LIN {X 50.548,Y -47.576,Z -199.936,A -90.000,B 90.000,C 0.000} C_DIS
LIN {X 49.783,Y -47.603,Z -202.584,A -90.000,B 90.000,C 0.000} C_DIS
LIN {X 49.593,Y -47.607,Z -203.194,A -90.000,B 90.000,C 0.000} C_DIS
LIN {X 48.332,Y -47.644,Z -207.156,A -90.000,B 90.000,C 0.000} C_DIS
LIN {X 47.582,Y -47.662,Z -209.460,A -90.000,B 90.000,C 0.000} C_DIS
LIN {X 47.233,Y -47.673,Z -210.498,A -90.000,B 90.000,C 0.000} C_DIS
LIN {X 46.703,Y -47.673,Z -212.067,A -90.000,B 90.000,C 0.000} C_DIS
LIN {X 46.008,Y -47.674,Z -214.062,A -90.000,B 90.000,C 0.000} C_DIS
LIN {X 45.274,Y -47.666,Z -216.296,A -90.000,B 90.000,C 0.000} C_DIS
LIN {X 44.970,Y -47.666,Z -217.223,A -90.000,B 90.000,C 0.000} C_DIS
LIN {X 44.923,Y -47.667,Z -217.335,A -90.000,B 90.000,C 0.000} C_DIS
LIN {X 44.486,Y -47.667,Z -218.383,A -90.000,B 90.000,C 0.000} C_DIS
LIN {X 43.526,Y -47.657,Z -220.833,A -90.000,B 90.000,C 0.000} C_DIS
LIN {X 42.934,Y -47.657,Z -222.345,A -90.000,B 90.000,C 0.000} C_DIS
LIN {X 42.807,Y -47.663,Z -222.577,A -90.000,B 90.000,C 0.000} C_DIS
LIN {X 42.638,Y -47.663,Z -222.882,A -90.000,B 90.000,C 0.000} C_DIS
LIN {X 41.300,Y -47.652,Z -225.431,A -90.000,B 90.000,C 0.000} C_DIS
LIN {X 40.291,Y -47.650,Z -227.357,A -90.000,B 90.000,C 0.000} C_DIS
LIN {X 40.021,Y -47.664,Z -227.703,A -90.000,B 90.000,C 0.000} C_DIS
LIN {X 39.850,Y -47.667,Z -227.921,A -90.000,B 90.000,C 0.000} C_DIS
LIN {X 37.302,Y -47.652,Z -231.289,A -90.000,B 90.000,C 0.000} C_DIS
LIN {X 36.746,Y -47.651,Z -232.025,A -90.000,B 90.000,C 0.000} C_DIS
LIN {X 36.686,Y -47.653,Z -232.080,A -90.000,B 90.000,C 0.000} C_DIS
LIN {X 36.061,Y -47.684,Z -232.614,A -90.000,B 90.000,C 0.000} C_DIS
LIN {X 35.829,Y -47.686,Z -232.809,A -90.000,B 90.000,C 0.000} C_DIS
LIN {X 35.506,Y -47.686,Z -233.081,A -90.000,B 90.000,C 0.000} C_DIS
LIN {X 34.289,Y -47.685,Z -234.104,A -90.000,B 90.000,C 0.000} C_DIS
LIN {X 33.544,Y -47.662,Z -234.725,A -90.000,B 90.000,C 0.000} C_DIS
LIN {X 31.821,Y -47.603,Z -236.201,A -90.000,B 90.000,C 0.000} C_DIS
LIN {X 31.643,Y -47.599,Z -236.332,A -90.000,B 90.000,C 0.000} C_DIS
LIN {X 30.851,Y -47.588,Z -236.838,A -90.000,B 90.000,C 0.000} C_DIS
LIN {X 30.642,Y -47.585,Z -236.965,A -90.000,B 90.000,C 0.000} C_DIS
LIN {X 29.999,Y -47.565,Z -237.355,A -90.000,B 90.000,C 0.000} C_DIS
LIN {X 26.309,Y -47.565,Z -238.632,A -90.000,B 90.000,C 0.000} C_DIS
LIN {X 26.101,Y -47.561,Z -238.703,A -90.000,B 90.000,C 0.000} C_DIS
LIN {X 25.572,Y -47.541,Z -238.883,A -90.000,B 90.000,C 0.000} C_DIS
LIN {X 24.943,Y -47.512,Z -239.098,A -90.000,B 90.000,C 0.000} C_DIS
LIN {X 24.543,Y -47.495,Z -239.210,A -90.000,B 90.000,C 0.000} C_DIS
LIN {X 24.462,Y -47.492,Z -239.233,A -90.000,B 90.000,C 0.000} C_DIS
LIN {X 24.387,Y -47.494,Z -239.257,A -90.000,B 90.000,C 0.000} C_DIS
LIN {X 24.313,Y -47.492,Z -239.283,A -90.000,B 90.000,C 0.000} C_DIS
LIN {X 24.239,Y -47.490,Z -239.311,A -90.000,B 90.000,C 0.000} C_DIS
LIN {X 24.093,Y -47.485,Z -239.376,A -90.000,B 90.000,C 0.000} C_DIS
LIN {X 23.947,Y -47.481,Z -239.382,A -90.000,B 90.000,C 0.000} C_DIS
LIN {X 23.875,Y -47.479,Z -239.388,A -90.000,B 90.000,C 0.000} C_DIS
LIN {X 23.732,Y -47.475,Z -239.409,A -90.000,B 90.000,C 0.000} C_DIS
LIN {X 23.592,Y -47.471,Z -239.439,A -90.000,B 90.000,C 0.000} C_DIS
LIN {X 23.385,Y -47.464,Z -239.496,A -90.000,B 90.000,C 0.000} C_DIS
LIN {X 23.249,Y -47.459,Z -239.542,A -90.000,B 90.000,C 0.000} C_DIS
LIN {X 23.115,Y -47.453,Z -239.594,A -90.000,B 90.000,C 0.000} C_DIS
LIN {X 22.916,Y -47.444,Z -239.681,A -90.000,B 90.000,C 0.000} C_DIS
LIN {X 22.655,Y -47.432,Z -239.810,A -90.000,B 90.000,C 0.000} C_DIS
LIN {X 22.008,Y -47.400,Z -240.160,A -90.000,B 90.000,C 0.000} C_DIS
LIN {X 21.748,Y -47.387,Z -240.295,A -90.000,B 90.000,C 0.000} C_DIS
LIN {X 21.484,Y -47.375,Z -240.419,A -90.000,B 90.000,C 0.000} C_DIS
LIN {X 21.350,Y -47.368,Z -240.477,A -90.000,B 90.000,C 0.000} C_DIS
LIN {X 21.215,Y -47.362,Z -240.528,A -90.000,B 90.000,C 0.000} C_DIS
LIN {X 21.078,Y -47.356,Z -240.571,A -90.000,B 90.000,C 0.000} C_DIS
LIN {X 21.009,Y -47.353,Z -240.590,A -90.000,B 90.000,C 0.000} C_DIS
LIN {X 20.940,Y -47.350,Z -240.606,A -90.000,B 90.000,C 0.000} C_DIS
LIN {X 20.839,Y -47.345,Z -240.621,A -90.000,B 90.000,C 0.000} C_DIS
LIN {X 20.661,Y -47.337,Z -240.664,A -90.000,B 90.000,C 0.000} C_DIS
LIN {X 20.513,Y -47.331,Z -240.694,A -90.000,B 90.000,C 0.000} C_DIS
LIN {X 20.361,Y -47.324,Z -240.716,A -90.000,B 90.000,C 0.000} C_DIS
LIN {X 20.284,Y -47.321,Z -240.723,A -90.000,B 90.000,C 0.000} C_DIS
LIN {X 20.127,Y -47.314,Z -240.729,A -90.000,B 90.000,C 0.000} C_DIS
LIN {X 20.049,Y -47.308,Z -240.727,A -90.000,B 90.000,C 0.000} C_DIS
LIN {X 19.691,Y -47.308,Z -240.706,A -90.000,B 90.000,C 0.000} C_DIS
LIN {X 19.298,Y -47.308,Z -240.660,A -90.000,B 90.000,C 0.000} C_DIS
LIN {X 19.221,Y -47.308,Z -240.617,A -90.000,B 90.000,C 0.000} C_DIS
LIN {X 17.099,Y -47.308,Z -237.044,A -90.000,B 90.000,C 0.000} C_DIS
LIN {X 17.057,Y -47.308,Z -236.966,A -90.000,B 90.000,C 0.000} C_DIS
LIN {X 17.047,Y -47.308,Z -236.943,A -90.000,B 90.000,C 0.000} C_DIS
LIN {X 16.984,Y -47.308,Z -236.487,A -90.000,B 90.000,C 0.000} C_DIS
LIN {X 16.973,Y -47.308,Z -236.308,A -90.000,B 90.000,C 0.000} C_DIS
LIN {X 17.928,Y -47.308,Z -231.443,A -90.000,B 90.000,C 0.000} C_DIS
LIN {X 17.967,Y -47.308,Z -231.268,A -90.000,B 90.000,C 0.000} C_DIS
LIN {X 19.365,Y -47.308,Z -226.787,A -90.000,B 90.000,C 0.000} C_DIS
LIN {X 19.696,Y -47.308,Z -226.007,A -90.000,B 90.000,C 0.000} C_DIS
LIN {X 20.442,Y -47.308,Z -224.463,A -90.000,B 90.000,C 0.000} C_DIS
LIN {X 22.215,Y -47.308,Z -221.029,A -90.000,B 90.000,C 0.000} C_DIS
LIN {X 24.188,Y -47.308,Z -217.425,A -90.000,B 90.000,C 0.000} C_DIS
LIN {X 24.824,Y -47.308,Z -216.161,A -90.000,B 90.000,C 0.000} C_DIS
LIN {X 26.477,Y -47.308,Z -213.204,A -90.000,B 90.000,C 0.000} C_DIS
LIN {X 27.332,Y -47.308,Z -211.400,A -90.000,B 90.000,C 0.000} C_DIS
LIN {X 28.292,Y -47.308,Z -209.670,A -90.000,B 90.000,C 0.000} C_DIS
LIN {X 29.492,Y -47.308,Z -206.852,A -90.000,B 90.000,C 0.000} C_DIS
LIN {X 29.913,Y -47.308,Z -206.062,A -90.000,B 90.000,C 0.000} C_DIS
LIN {X 30.848,Y -47.308,Z -203.410,A -90.000,B 90.000,C 0.000} C_DIS
LIN {X 31.216,Y -47.308,Z -202.524,A -90.000,B 90.000,C 0.000} C_DIS
LIN {X 31.238,Y -47.308,Z -202.440,A -90.000,B 90.000,C 0.000} C_DIS
LIN {X 32.486,Y -47.308,Z -199.249,A -90.000,B 90.000,C 0.000} C_DIS
LIN {X 32.612,Y -47.308,Z -198.488,A -90.000,B 90.000,C 0.000} C_DIS
LIN {X 32.650,Y -47.308,Z -198.313,A -90.000,B 90.000,C 0.000} C_DIS
LIN {X 33.456,Y -47.308,Z -196.184,A -90.000,B 90.000,C 0.000} C_DIS
LIN {X 33.655,Y -47.308,Z -194.664,A -90.000,B 90.000,C 0.000} C_DIS
LIN {X 33.694,Y -47.308,Z -194.489,A -90.000,B 90.000,C 0.000} C_DIS
LIN {X 34.211,Y -47.308,Z -193.297,A -90.000,B 90.000,C 0.000} C_DIS
LIN {X 34.763,Y -47.308,Z -191.054,A -90.000,B 90.000,C 0.000} C_DIS
LIN {X 34.848,Y -47.308,Z -190.896,A -90.000,B 90.000,C 0.000} C_DIS
LIN {X 36.168,Y -47.308,Z -188.741,A -90.000,B 90.000,C 0.000} C_DIS
LIN {X 36.650,Y -47.308,Z -187.989,A -90.000,B 90.000,C 0.000} C_DIS
LIN {X 37.823,Y -47.308,Z -186.759,A -90.000,B 90.000,C 0.000} C_DIS
LIN {X 38.833,Y -47.308,Z -185.482,A -90.000,B 90.000,C 0.000} C_DIS
LIN {X 38.959,Y -47.308,Z -185.354,A -90.000,B 90.000,C 0.000} C_DIS
LIN {X 39.438,Y -47.308,Z -184.917,A -90.000,B 90.000,C 0.000} C_DIS
LIN {X 40.740,Y -47.308,Z -183.333,A -90.000,B 90.000,C 0.000} C_DIS
LIN {X 40.875,Y -47.308,Z -183.194,A -90.000,B 90.000,C 0.000} C_DIS
LIN {X 40.967,Y -47.308,Z -183.111,A -90.000,B 90.000,C 0.000} C_DIS
LIN {X 41.001,Y -47.308,Z -183.078,A -90.000,B 90.000,C 0.000} C_DIS
LIN {X 42.416,Y -47.308,Z -181.743,A -90.000,B 90.000,C 0.000} C_DIS
LIN {X 42.967,Y -47.308,Z -181.080,A -90.000,B 90.000,C 0.000} C_DIS
LIN {X 43.744,Y -47.308,Z -180.119,A -90.000,B 90.000,C 0.000} C_DIS
LIN {X 44.641,Y -47.308,Z -178.883,A -90.000,B 90.000,C 0.000} C_DIS
LIN {X 45.026,Y -47.308,Z -178.318,A -90.000,B 90.000,C 0.000} C_DIS
LIN {X 46.161,Y -47.308,Z -176.577,A -90.000,B 90.000,C 0.000} C_DIS
LIN {X 46.268,Y -47.308,Z -176.406,A -90.000,B 90.000,C 0.000} C_DIS
LIN {X 46.785,Y -47.308,Z -175.538,A -90.000,B 90.000,C 0.000} C_DIS
LIN {X 47.568,Y -47.308,Z -174.267,A -90.000,B 90.000,C 0.000} C_DIS
LIN {X 47.989,Y -47.308,Z -173.536,A -90.000,B 90.000,C 0.000} C_DIS
LIN {X 48.041,Y -47.308,Z -173.464,A -90.000,B 90.000,C 0.000} C_DIS
LIN {X 49.321,Y -47.308,Z -172.666,A -90.000,B 90.000,C 0.000} C_DIS
LIN {X 50.521,Y -47.308,Z -171.855,A -90.000,B 90.000,C 0.000} C_DIS
LIN {X 51.142,Y -47.308,Z -171.455,A -90.000,B 90.000,C 0.000} C_DIS
LIN {X 51.886,Y -47.308,Z -170.509,A -90.000,B 90.000,C 0.000} C_DIS
LIN {X 52.063,Y -47.308,Z -170.387,A -90.000,B 90.000,C 0.000} C_DIS
LIN {X 52.122,Y -47.308,Z -170.550,A -90.000,B 90.000,C 0.000} C_DIS
LIN {X 52.146,Y -47.308,Z -170.635,A -90.000,B 90.000,C 0.000} C_DIS
LIN {X 51.989,Y -47.308,Z -172.198,A -90.000,B 90.000,C 0.000} C_DIS
LIN {X 51.995,Y -47.308,Z -172.668,A -90.000,B 90.000,C 0.000} C_DIS
LIN {X 51.980,Y -47.308,Z -175.146,A -90.000,B 90.000,C 0.000} C_DIS
LIN {X 52.499,Y -47.308,Z -177.649,A -90.000,B 90.000,C 0.000} C_DIS
LIN {X 52.544,Y -47.308,Z -177.979,A -90.000,B 90.000,C 0.000} C_DIS
LIN {X 52.649,Y -47.308,Z -178.226,A -90.000,B 90.000,C 0.000} C_DIS
LIN {X 52.673,Y -47.308,Z -178.312,A -90.000,B 90.000,C 0.000} C_DIS
LIN {X 52.771,Y -47.308,Z -179.420,A -90.000,B 90.000,C 0.000} C_DIS
LIN {X 52.804,Y -47.308,Z -180.560,A -90.000,B 90.000,C 0.000} C_DIS
LIN {X 52.909,Y -47.308,Z -181.087,A -90.000,B 90.000,C 0.000} C_DIS
LIN {X 52.928,Y -47.308,Z -181.222,A -90.000,B 90.000,C 0.000} C_DIS
LIN {X 53.150,Y -47.308,Z -183.107,A -90.000,B 90.000,C 0.000} C_DIS
LIN {X 53.819,Y -47.308,Z -185.717,A -90.000,B 90.000,C 0.000} C_DIS
LIN {X 53.836,Y -47.308,Z -185.790,A -90.000,B 90.000,C 0.000} C_DIS
LIN {X 53.860,Y -47.308,Z -185.967,A -90.000,B 90.000,C 0.000} C_DIS
LIN {X 53.930,Y -47.308,Z -188.587,A -90.000,B 90.000,C 0.000} C_DIS
LIN {X 53.954,Y -47.308,Z -189.753,A -90.000,B 90.000,C 0.000} C_DIS
LIN {X 53.918,Y -47.308,Z -191.505,A -90.000,B 90.000,C 0.000} C_DIS
LIN {X 53.761,Y -47.308,Z -194.195,A -90.000,B 90.000,C 0.000} C_DIS
LIN {X 53.699,Y -47.308,Z -194.926,A -90.000,B 90.000,C 0.000} C_DIS
LIN {X 53.629,Y -47.308,Z -195.338,A -90.000,B 90.000,C 0.000} C_DIS
LIN {X 53.425,Y -47.308,Z -196.821,A -90.000,B 90.000,C 0.000} C_DIS
LIN {X 52.961,Y -47.308,Z -198.727,A -90.000,B 90.000,C 0.000} C_DIS
LIN {X 52.919,Y -47.308,Z -198.878,A -90.000,B 90.000,C 0.000} C_DIS
LIN {X 51.671,Y -47.308,Z -203.173,A -90.000,B 90.000,C 0.000} C_DIS
LIN {X 51.479,Y -47.308,Z -203.790,A -90.000,B 90.000,C 0.000} C_DIS
LIN {X 50.206,Y -47.308,Z -207.769,A -90.000,B 90.000,C 0.000} C_DIS
LIN {X 49.447,Y -47.308,Z -210.090,A -90.000,B 90.000,C 0.000} C_DIS
LIN {X 48.560,Y -47.308,Z -212.715,A -90.000,B 90.000,C 0.000} C_DIS
LIN {X 47.876,Y -47.308,Z -214.675,A -90.000,B 90.000,C 0.000} C_DIS
LIN {X 46.815,Y -47.308,Z -217.909,A -90.000,B 90.000,C 0.000} C_DIS
LIN {X 46.302,Y -47.308,Z -219.140,A -90.000,B 90.000,C 0.000} C_DIS
LIN {X 44.720,Y -47.308,Z -223.185,A -90.000,B 90.000,C 0.000} C_DIS
LIN {X 44.360,Y -47.308,Z -223.835,A -90.000,B 90.000,C 0.000} C_DIS
LIN {X 41.992,Y -47.308,Z -228.356,A -90.000,B 90.000,C 0.000} C_DIS
LIN {X 41.894,Y -47.308,Z -228.506,A -90.000,B 90.000,C 0.000} C_DIS
LIN {X 41.395,Y -47.308,Z -229.139,A -90.000,B 90.000,C 0.000} C_DIS
LIN {X 38.208,Y -47.308,Z -233.359,A -90.000,B 90.000,C 0.000} C_DIS
LIN {X 37.985,Y -47.308,Z -233.562,A -90.000,B 90.000,C 0.000} C_DIS
LIN {X 34.811,Y -47.308,Z -236.231,A -90.000,B 90.000,C 0.000} C_DIS
LIN {X 33.058,Y -47.308,Z -237.747,A -90.000,B 90.000,C 0.000} C_DIS
LIN {X 32.767,Y -47.308,Z -237.962,A -90.000,B 90.000,C 0.000} C_DIS
LIN {X 31.901,Y -47.308,Z -238.517,A -90.000,B 90.000,C 0.000} C_DIS
LIN {X 30.925,Y -47.308,Z -239.114,A -90.000,B 90.000,C 0.000} C_DIS
LIN {X 30.762,Y -47.308,Z -239.190,A -90.000,B 90.000,C 0.000} C_DIS
LIN {X 25.551,Y -47.308,Z -240.992,A -90.000,B 90.000,C 0.000} C_DIS
LIN {X 24.857,Y -47.308,Z -241.192,A -90.000,B 90.000,C 0.000} C_DIS
LIN {X 24.342,Y -47.308,Z -241.346,A -90.000,B 90.000,C 0.000} C_DIS
LIN {X 24.165,Y -47.308,Z -241.375,A -90.000,B 90.000,C 0.000} C_DIS
LIN {X 23.987,Y -47.308,Z -241.353,A -90.000,B 90.000,C 0.000} C_DIS
LIN {X 20.879,Y -47.308,Z -240.774,A -90.000,B 90.000,C 0.000} C_DIS
LIN {X 20.049,Y -47.308,Z -240.727,A -90.000,B 90.000,C 0.000} C_DIS
LIN {X 20.049,Y -60.000,Z -240.727,A -90.000,B 90.000,C 0.000} C_DIS
LIN {X 38.586,Y -60.000,Z -66.482,A -90.000,B 90.000,C 0.000} C_DIS
LIN {X 38.586,Y -46.332,Z -66.482,A -90.000,B 90.000,C 0.000} C_DIS
LIN {X 38.743,Y -46.408,Z -65.766,A -90.000,B 90.000,C 0.000} C_DIS
LIN {X 38.814,Y -46.447,Z -65.441,A -90.000,B 90.000,C 0.000} C_DIS
LIN {X 38.832,Y -46.453,Z -65.361,A -90.000,B 90.000,C 0.000} C_DIS
LIN {X 39.021,Y -46.481,Z -65.010,A -90.000,B 90.000,C 0.000} C_DIS
LIN {X 39.070,Y -46.483,Z -64.924,A -90.000,B 90.000,C 0.000} C_DIS
LIN {X 39.296,Y -46.478,Z -64.552,A -90.000,B 90.000,C 0.000} C_DIS
LIN {X 39.367,Y -46.470,Z -64.429,A -90.000,B 90.000,C 0.000} C_DIS
LIN {X 39.510,Y -46.448,Z -64.171,A -90.000,B 90.000,C 0.000} C_DIS
LIN {X 39.538,Y -46.445,Z -64.120,A -90.000,B 90.000,C 0.000} C_DIS
LIN {X 39.628,Y -46.438,Z -63.976,A -90.000,B 90.000,C 0.000} C_DIS
LIN {X 39.829,Y -46.434,Z -63.758,A -90.000,B 90.000,C 0.000} C_DIS
LIN {X 39.847,Y -46.433,Z -63.739,A -90.000,B 90.000,C 0.000} C_DIS
LIN {X 39.991,Y -46.429,Z -63.625,A -90.000,B 90.000,C 0.000} C_DIS
LIN {X 40.169,Y -46.420,Z -63.488,A -90.000,B 90.000,C 0.000} C_DIS
LIN {X 40.456,Y -46.402,Z -63.249,A -90.000,B 90.000,C 0.000} C_DIS
LIN {X 40.544,Y -46.395,Z -63.177,A -90.000,B 90.000,C 0.000} C_DIS
LIN {X 40.546,Y -46.395,Z -63.180,A -90.000,B 90.000,C 0.000} C_DIS
LIN {X 40.725,Y -46.409,Z -63.544,A -90.000,B 90.000,C 0.000} C_DIS
LIN {X 40.761,Y -46.412,Z -63.625,A -90.000,B 90.000,C 0.000} C_DIS
LIN {X 40.662,Y -46.455,Z -64.217,A -90.000,B 90.000,C 0.000} C_DIS
LIN {X 40.562,Y -46.497,Z -64.813,A -90.000,B 90.000,C 0.000} C_DIS
LIN {X 40.372,Y -46.518,Z -65.066,A -90.000,B 90.000,C 0.000} C_DIS
LIN {X 40.250,Y -46.525,Z -65.224,A -90.000,B 90.000,C 0.000} C_DIS
LIN {X 40.139,Y -46.523,Z -65.365,A -90.000,B 90.000,C 0.000} C_DIS
LIN {X 39.973,Y -46.509,Z -65.573,A -90.000,B 90.000,C 0.000} C_DIS
LIN {X 39.871,Y -46.497,Z -65.699,A -90.000,B 90.000,C 0.000} C_DIS
LIN {X 39.701,Y -46.467,Z -65.906,A -90.000,B 90.000,C 0.000} C_DIS
LIN {X 39.672,Y -46.462,Z -65.936,A -90.000,B 90.000,C 0.000} C_DIS
LIN {X 39.637,Y -46.457,Z -65.966,A -90.000,B 90.000,C 0.000} C_DIS
LIN {X 39.426,Y -46.430,Z -66.104,A -90.000,B 90.000,C 0.000} C_DIS
LIN {X 39.258,Y -46.405,Z -66.212,A -90.000,B 90.000,C 0.000} C_DIS
LIN {X 38.910,Y -46.357,Z -66.394,A -90.000,B 90.000,C 0.000} C_DIS
LIN {X 38.817,Y -46.347,Z -66.419,A -90.000,B 90.000,C 0.000} C_DIS
LIN {X 38.586,Y -46.332,Z -66.482,A -90.000,B 90.000,C 0.000} C_DIS
LIN {X 38.730,Y -46.403,Z -65.860,A -90.000,B 90.000,C 0.000} C_DIS
LIN {X 38.763,Y -46.422,Z -65.690,A -90.000,B 90.000,C 0.000} C_DIS
LIN {X 38.780,Y -46.436,Z -65.558,A -90.000,B 90.000,C 0.000} C_DIS
LIN {X 38.820,Y -46.445,Z -65.487,A -90.000,B 90.000,C 0.000} C_DIS
LIN {X 38.866,Y -46.457,Z -65.390,A -90.000,B 90.000,C 0.000} C_DIS
LIN {X 38.895,Y -46.465,Z -65.310,A -90.000,B 90.000,C 0.000} C_DIS
LIN {X 38.902,Y -46.468,Z -65.275,A -90.000,B 90.000,C 0.000} C_DIS
LIN {X 38.901,Y -46.469,Z -65.244,A -90.000,B 90.000,C 0.000} C_DIS
LIN {X 38.899,Y -46.470,Z -65.230,A -90.000,B 90.000,C 0.000} C_DIS
LIN {X 38.886,Y -46.470,Z -65.204,A -90.000,B 90.000,C 0.000} C_DIS
LIN {X 38.865,Y -46.470,Z -65.181,A -90.000,B 90.000,C 0.000} C_DIS
LIN {X 38.838,Y -46.469,Z -65.136,A -90.000,B 90.000,C 0.000} C_DIS
LIN {X 38.805,Y -46.468,Z -65.095,A -90.000,B 90.000,C 0.000} C_DIS
LIN {X 38.773,Y -46.466,Z -65.065,A -90.000,B 90.000,C 0.000} C_DIS
LIN {X 38.722,Y -46.462,Z -65.036,A -90.000,B 90.000,C 0.000} C_DIS
LIN {X 38.546,Y -46.448,Z -64.983,A -90.000,B 90.000,C 0.000} C_DIS
LIN {X 38.421,Y -46.433,Z -64.934,A -90.000,B 90.000,C 0.000} C_DIS
LIN {X 38.302,Y -46.415,Z -65.036,A -90.000,B 90.000,C 0.000} C_DIS
LIN {X 38.274,Y -46.410,Z -65.056,A -90.000,B 90.000,C 0.000} C_DIS
LIN {X 38.217,Y -46.400,Z -65.089,A -90.000,B 90.000,C 0.000} C_DIS
LIN {X 38.174,Y -46.394,Z -65.107,A -90.000,B 90.000,C 0.000} C_DIS
LIN {X 38.113,Y -46.386,Z -65.120,A -90.000,B 90.000,C 0.000} C_DIS
LIN {X 38.073,Y -46.381,Z -65.126,A -90.000,B 90.000,C 0.000} C_DIS
LIN {X 37.996,Y -46.371,Z -65.130,A -90.000,B 90.000,C 0.000} C_DIS
LIN {X 37.958,Y -46.366,Z -65.128,A -90.000,B 90.000,C 0.000} C_DIS
LIN {X 37.887,Y -46.356,Z -65.115,A -90.000,B 90.000,C 0.000} C_DIS
LIN {X 37.852,Y -46.352,Z -65.105,A -90.000,B 90.000,C 0.000} C_DIS
LIN {X 37.786,Y -46.342,Z -65.076,A -90.000,B 90.000,C 0.000} C_DIS
LIN {X 37.754,Y -46.338,Z -65.058,A -90.000,B 90.000,C 0.000} C_DIS
LIN {X 37.693,Y -46.328,Z -65.015,A -90.000,B 90.000,C 0.000} C_DIS
LIN {X 37.637,Y -46.318,Z -64.962,A -90.000,B 90.000,C 0.000} C_DIS
LIN {X 37.584,Y -46.308,Z -64.900,A -90.000,B 90.000,C 0.000} C_DIS
LIN {X 37.536,Y -46.296,Z -64.828,A -90.000,B 90.000,C 0.000} C_DIS
LIN {X 37.488,Y -46.284,Z -64.747,A -90.000,B 90.000,C 0.000} C_DIS
LIN {X 37.470,Y -46.279,Z -64.714,A -90.000,B 90.000,C 0.000} C_DIS
LIN {X 37.452,Y -46.272,Z -64.660,A -90.000,B 90.000,C 0.000} C_DIS
LIN {X 37.437,Y -46.260,Z -64.573,A -90.000,B 90.000,C 0.000} C_DIS
LIN {X 37.429,Y -46.248,Z -64.480,A -90.000,B 90.000,C 0.000} C_DIS
LIN {X 37.432,Y -46.229,Z -64.332,A -90.000,B 90.000,C 0.000} C_DIS
LIN {X 37.443,Y -46.216,Z -64.229,A -90.000,B 90.000,C 0.000} C_DIS
LIN {X 37.460,Y -46.202,Z -64.122,A -90.000,B 90.000,C 0.000} C_DIS
LIN {X 37.484,Y -46.187,Z -64.012,A -90.000,B 90.000,C 0.000} C_DIS
LIN {X 37.516,Y -46.172,Z -63.902,A -90.000,B 90.000,C 0.000} C_DIS
LIN {X 37.554,Y -46.157,Z -63.791,A -90.000,B 90.000,C 0.000} C_DIS
LIN {X 37.596,Y -46.142,Z -63.678,A -90.000,B 90.000,C 0.000} C_DIS
LIN {X 37.713,Y -46.102,Z -63.395,A -90.000,B 90.000,C 0.000} C_DIS
LIN {X 37.790,Y -46.078,Z -63.229,A -90.000,B 90.000,C 0.000} C_DIS
LIN {X 37.846,Y -46.063,Z -63.124,A -90.000,B 90.000,C 0.000} C_DIS
LIN {X 37.993,Y -46.061,Z -62.882,A -90.000,B 90.000,C 0.000} C_DIS
LIN {X 38.118,Y -46.066,Z -62.715,A -90.000,B 90.000,C 0.000} C_DIS
LIN {X 38.400,Y -46.084,Z -62.403,A -90.000,B 90.000,C 0.000} C_DIS
LIN {X 38.485,Y -46.085,Z -62.311,A -90.000,B 90.000,C 0.000} C_DIS
LIN {X 38.586,Y -46.089,Z -62.224,A -90.000,B 90.000,C 0.000} C_DIS
LIN {X 38.789,Y -46.087,Z -62.063,A -90.000,B 90.000,C 0.000} C_DIS
LIN {X 38.911,Y -46.079,Z -61.970,A -90.000,B 90.000,C 0.000} C_DIS
LIN {X 38.995,Y -46.071,Z -61.902,A -90.000,B 90.000,C 0.000} C_DIS
LIN {X 39.206,Y -46.041,Z -61.731,A -90.000,B 90.000,C 0.000} C_DIS
LIN {X 39.476,Y -45.996,Z -61.513,A -90.000,B 90.000,C 0.000} C_DIS
LIN {X 39.640,Y -45.971,Z -61.387,A -90.000,B 90.000,C 0.000} C_DIS
LIN {X 39.702,Y -45.965,Z -61.351,A -90.000,B 90.000,C 0.000} C_DIS
LIN {X 39.744,Y -45.964,Z -61.336,A -90.000,B 90.000,C 0.000} C_DIS
LIN {X 39.940,Y -45.968,Z -61.275,A -90.000,B 90.000,C 0.000} C_DIS
LIN {X 40.138,Y -45.968,Z -61.215,A -90.000,B 90.000,C 0.000} C_DIS
LIN {X 40.210,Y -45.969,Z -61.197,A -90.000,B 90.000,C 0.000} C_DIS
LIN {X 40.415,Y -45.962,Z -61.149,A -90.000,B 90.000,C 0.000} C_DIS
LIN {X 40.526,Y -45.957,Z -61.124,A -90.000,B 90.000,C 0.000} C_DIS
LIN {X 40.635,Y -45.948,Z -61.096,A -90.000,B 90.000,C 0.000} C_DIS
LIN {X 40.700,Y -45.947,Z -61.093,A -90.000,B 90.000,C 0.000} C_DIS
LIN {X 40.722,Y -45.946,Z -61.095,A -90.000,B 90.000,C 0.000} C_DIS
LIN {X 40.933,Y -45.948,Z -61.145,A -90.000,B 90.000,C 0.000} C_DIS
LIN {X 41.055,Y -45.946,Z -61.174,A -90.000,B 90.000,C 0.000} C_DIS
LIN {X 41.403,Y -45.927,Z -61.265,A -90.000,B 90.000,C 0.000} C_DIS
LIN {X 41.663,Y -45.913,Z -61.345,A -90.000,B 90.000,C 0.000} C_DIS
LIN {X 41.709,Y -45.912,Z -61.366,A -90.000,B 90.000,C 0.000} C_DIS
LIN {X 41.741,Y -45.918,Z -61.402,A -90.000,B 90.000,C 0.000} C_DIS
LIN {X 41.859,Y -45.950,Z -61.574,A -90.000,B 90.000,C 0.000} C_DIS
LIN {X 42.116,Y -46.026,Z -61.976,A -90.000,B 90.000,C 0.000} C_DIS
LIN {X 42.161,Y -46.038,Z -62.045,A -90.000,B 90.000,C 0.000} C_DIS
LIN {X 42.276,Y -46.064,Z -62.230,A -90.000,B 90.000,C 0.000} C_DIS
LIN {X 42.315,Y -46.075,Z -62.304,A -90.000,B 90.000,C 0.000} C_DIS
LIN {X 42.375,Y -46.088,Z -62.420,A -90.000,B 90.000,C 0.000} C_DIS
LIN {X 42.443,Y -46.100,Z -62.555,A -90.000,B 90.000,C 0.000} C_DIS
LIN {X 42.519,Y -46.106,Z -62.714,A -90.000,B 90.000,C 0.000} C_DIS
LIN {X 42.561,Y -46.108,Z -62.802,A -90.000,B 90.000,C 0.000} C_DIS
LIN {X 42.601,Y -46.108,Z -62.900,A -90.000,B 90.000,C 0.000} C_DIS
LIN {X 42.677,Y -46.103,Z -63.092,A -90.000,B 90.000,C 0.000} C_DIS
LIN {X 42.766,Y -46.084,Z -63.342,A -90.000,B 90.000,C 0.000} C_DIS
LIN {X 42.777,Y -46.080,Z -63.401,A -90.000,B 90.000,C 0.000} C_DIS
LIN {X 42.782,Y -46.077,Z -63.475,A -90.000,B 90.000,C 0.000} C_DIS
LIN {X 42.770,Y -46.079,Z -63.601,A -90.000,B 90.000,C 0.000} C_DIS
LIN {X 42.470,Y -46.135,Z -65.317,A -90.000,B 90.000,C 0.000} C_DIS
LIN {X 42.459,Y -46.135,Z -65.378,A -90.000,B 90.000,C 0.000} C_DIS
LIN {X 42.420,Y -46.138,Z -65.540,A -90.000,B 90.000,C 0.000} C_DIS
LIN {X 42.387,Y -46.141,Z -65.627,A -90.000,B 90.000,C 0.000} C_DIS
LIN {X 42.325,Y -46.147,Z -65.741,A -90.000,B 90.000,C 0.000} C_DIS
LIN {X 42.249,Y -46.155,Z -65.848,A -90.000,B 90.000,C 0.000} C_DIS
LIN {X 42.116,Y -46.163,Z -66.027,A -90.000,B 90.000,C 0.000} C_DIS
LIN {X 41.951,Y -46.159,Z -66.242,A -90.000,B 90.000,C 0.000} C_DIS
LIN {X 41.233,Y -46.093,Z -67.137,A -90.000,B 90.000,C 0.000} C_DIS
LIN {X 41.182,Y -46.090,Z -67.197,A -90.000,B 90.000,C 0.000} C_DIS
LIN {X 41.068,Y -46.082,Z -67.320,A -90.000,B 90.000,C 0.000} C_DIS
LIN {X 40.966,Y -46.079,Z -67.412,A -90.000,B 90.000,C 0.000} C_DIS
LIN {X 40.870,Y -46.074,Z -67.498,A -90.000,B 90.000,C 0.000} C_DIS
LIN {X 40.702,Y -46.072,Z -67.617,A -90.000,B 90.000,C 0.000} C_DIS
LIN {X 40.358,Y -46.077,Z -67.850,A -90.000,B 90.000,C 0.000} C_DIS
LIN {X 40.275,Y -46.075,Z -67.904,A -90.000,B 90.000,C 0.000} C_DIS
LIN {X 39.841,Y -46.072,Z -68.141,A -90.000,B 90.000,C 0.000} C_DIS
LIN {X 39.694,Y -46.064,Z -68.218,A -90.000,B 90.000,C 0.000} C_DIS
LIN {X 39.587,Y -46.061,Z -68.259,A -90.000,B 90.000,C 0.000} C_DIS
LIN {X 39.348,Y -46.052,Z -68.324,A -90.000,B 90.000,C 0.000} C_DIS
LIN {X 39.093,Y -46.030,Z -68.393,A -90.000,B 90.000,C 0.000} C_DIS
LIN {X 38.750,Y -45.982,Z -68.480,A -90.000,B 90.000,C 0.000} C_DIS
LIN {X 38.431,Y -45.935,Z -68.561,A -90.000,B 90.000,C 0.000} C_DIS
LIN {X 38.390,Y -45.930,Z -68.567,A -90.000,B 90.000,C 0.000} C_DIS
LIN {X 38.315,Y -45.928,Z -68.559,A -90.000,B 90.000,C 0.000} C_DIS
LIN {X 38.090,Y -45.923,Z -68.524,A -90.000,B 90.000,C 0.000} C_DIS
LIN {X 37.725,Y -45.920,Z -68.469,A -90.000,B 90.000,C 0.000} C_DIS
LIN {X 37.590,Y -45.912,Z -68.445,A -90.000,B 90.000,C 0.000} C_DIS
LIN {X 37.554,Y -45.911,Z -68.436,A -90.000,B 90.000,C 0.000} C_DIS
LIN {X 37.538,Y -45.911,Z -68.429,A -90.000,B 90.000,C 0.000} C_DIS
LIN {X 37.495,Y -45.913,Z -68.402,A -90.000,B 90.000,C 0.000} C_DIS
LIN {X 37.296,Y -45.911,Z -68.274,A -90.000,B 90.000,C 0.000} C_DIS
LIN {X 37.060,Y -45.898,Z -68.115,A -90.000,B 90.000,C 0.000} C_DIS
LIN {X 36.967,Y -45.888,Z -68.051,A -90.000,B 90.000,C 0.000} C_DIS
LIN {X 36.949,Y -45.892,Z -68.012,A -90.000,B 90.000,C 0.000} C_DIS
LIN {X 36.896,Y -45.909,Z -67.865,A -90.000,B 90.000,C 0.000} C_DIS
LIN {X 36.779,Y -45.952,Z -67.497,A -90.000,B 90.000,C 0.000} C_DIS
LIN {X 36.742,Y -45.965,Z -67.383,A -90.000,B 90.000,C 0.000} C_DIS
LIN {X 36.703,Y -45.986,Z -67.217,A -90.000,B 90.000,C 0.000} C_DIS
LIN {X 36.663,Y -46.003,Z -67.034,A -90.000,B 90.000,C 0.000} C_DIS
LIN {X 36.619,Y -46.010,Z -66.817,A -90.000,B 90.000,C 0.000} C_DIS
LIN {X 36.605,Y -46.009,Z -66.741,A -90.000,B 90.000,C 0.000} C_DIS
LIN {X 36.594,Y -46.011,Z -66.582,A -90.000,B 90.000,C 0.000} C_DIS
LIN {X 36.586,Y -46.010,Z -66.404,A -90.000,B 90.000,C 0.000} C_DIS
LIN {X 36.592,Y -46.011,Z -66.336,A -90.000,B 90.000,C 0.000} C_DIS
LIN {X 36.702,Y -46.036,Z -65.852,A -90.000,B 90.000,C 0.000} C_DIS
LIN {X 36.972,Y -46.085,Z -64.686,A -90.000,B 90.000,C 0.000} C_DIS
LIN {X 36.995,Y -46.087,Z -64.626,A -90.000,B 90.000,C 0.000} C_DIS
LIN {X 37.095,Y -46.098,Z -64.435,A -90.000,B 90.000,C 0.000} C_DIS
LIN {X 37.211,Y -46.098,Z -64.224,A -90.000,B 90.000,C 0.000} C_DIS
LIN {X 37.362,Y -46.089,Z -63.960,A -90.000,B 90.000,C 0.000} C_DIS
LIN {X 37.625,Y -46.072,Z -63.530,A -90.000,B 90.000,C 0.000} C_DIS
LIN {X 37.831,Y -46.063,Z -63.149,A -90.000,B 90.000,C 0.000} C_DIS
LIN {X 37.846,Y -46.063,Z -63.124,A -90.000,B 90.000,C 0.000} C_DIS
LIN {X 37.923,Y -46.062,Z -62.986,A -90.000,B 90.000,C 0.000} C_DIS
LIN {X 38.068,Y -46.055,Z -62.706,A -90.000,B 90.000,C 0.000} C_DIS
LIN {X 38.143,Y -46.051,Z -62.570,A -90.000,B 90.000,C 0.000} C_DIS
LIN {X 38.403,Y -46.003,Z -62.012,A -90.000,B 90.000,C 0.000} C_DIS
LIN {X 38.435,Y -45.992,Z -61.943,A -90.000,B 90.000,C 0.000} C_DIS
LIN {X 38.522,Y -45.947,Z -61.735,A -90.000,B 90.000,C 0.000} C_DIS
LIN {X 38.625,Y -45.886,Z -61.448,A -90.000,B 90.000,C 0.000} C_DIS
LIN {X 38.720,Y -45.824,Z -61.159,A -90.000,B 90.000,C 0.000} C_DIS
LIN {X 38.807,Y -45.761,Z -60.861,A -90.000,B 90.000,C 0.000} C_DIS
LIN {X 39.043,Y -45.630,Z -60.256,A -90.000,B 90.000,C 0.000} C_DIS
LIN {X 39.103,Y -45.601,Z -60.125,A -90.000,B 90.000,C 0.000} C_DIS
LIN {X 39.186,Y -45.565,Z -59.968,A -90.000,B 90.000,C 0.000} C_DIS
LIN {X 39.232,Y -45.549,Z -59.900,A -90.000,B 90.000,C 0.000} C_DIS
LIN {X 39.345,Y -45.513,Z -59.766,A -90.000,B 90.000,C 0.000} C_DIS
LIN {X 39.512,Y -45.467,Z -59.613,A -90.000,B 90.000,C 0.000} C_DIS
LIN {X 39.671,Y -45.426,Z -59.487,A -90.000,B 90.000,C 0.000} C_DIS
LIN {X 39.790,Y -45.398,Z -59.416,A -90.000,B 90.000,C 0.000} C_DIS
LIN {X 39.918,Y -45.370,Z -59.353,A -90.000,B 90.000,C 0.000} C_DIS
LIN {X 40.055,Y -45.340,Z -59.299,A -90.000,B 90.000,C 0.000} C_DIS
LIN {X 40.204,Y -45.308,Z -59.256,A -90.000,B 90.000,C 0.000} C_DIS
LIN {X 40.369,Y -45.308,Z -59.218,A -90.000,B 90.000,C 0.000} C_DIS
LIN {X 40.385,Y -45.308,Z -59.214,A -90.000,B 90.000,C 0.000} C_DIS
LIN {X 40.704,Y -45.308,Z -59.191,A -90.000,B 90.000,C 0.000} C_DIS
LIN {X 41.022,Y -45.308,Z -59.218,A -90.000,B 90.000,C 0.000} C_DIS
LIN {X 41.574,Y -45.308,Z -59.349,A -90.000,B 90.000,C 0.000} C_DIS
LIN {X 41.885,Y -45.308,Z -59.425,A -90.000,B 90.000,C 0.000} C_DIS
LIN {X 42.302,Y -45.308,Z -59.546,A -90.000,B 90.000,C 0.000} C_DIS
LIN {X 42.588,Y -45.308,Z -59.667,A -90.000,B 90.000,C 0.000} C_DIS
LIN {X 42.795,Y -45.308,Z -59.795,A -90.000,B 90.000,C 0.000} C_DIS
LIN {X 42.850,Y -45.308,Z -59.833,A -90.000,B 90.000,C 0.000} C_DIS
LIN {X 43.035,Y -45.308,Z -59.992,A -90.000,B 90.000,C 0.000} C_DIS
LIN {X 43.083,Y -45.308,Z -60.038,A -90.000,B 90.000,C 0.000} C_DIS
LIN {X 43.241,Y -45.308,Z -60.224,A -90.000,B 90.000,C 0.000} C_DIS
LIN {X 43.327,Y -45.308,Z -60.342,A -90.000,B 90.000,C 0.000} C_DIS
LIN {X 43.493,Y -45.308,Z -60.615,A -90.000,B 90.000,C 0.000} C_DIS
LIN {X 43.927,Y -45.308,Z -61.387,A -90.000,B 90.000,C 0.000} C_DIS
LIN {X 44.241,Y -45.308,Z -62.068,A -90.000,B 90.000,C 0.000} C_DIS
LIN {X 44.334,Y -45.308,Z -62.293,A -90.000,B 90.000,C 0.000} C_DIS
LIN {X 44.465,Y -45.308,Z -62.620,A -90.000,B 90.000,C 0.000} C_DIS
LIN {X 44.533,Y -45.308,Z -62.804,A -90.000,B 90.000,C 0.000} C_DIS
LIN {X 44.566,Y -45.308,Z -62.941,A -90.000,B 90.000,C 0.000} C_DIS
LIN {X 44.608,Y -45.308,Z -63.133,A -90.000,B 90.000,C 0.000} C_DIS
LIN {X 44.633,Y -45.308,Z -63.470,A -90.000,B 90.000,C 0.000} C_DIS
LIN {X 44.632,Y -45.308,Z -63.528,A -90.000,B 90.000,C 0.000} C_DIS
LIN {X 44.598,Y -45.308,Z -63.864,A -90.000,B 90.000,C 0.000} C_DIS
LIN {X 44.239,Y -45.308,Z -65.762,A -90.000,B 90.000,C 0.000} C_DIS
LIN {X 44.159,Y -45.308,Z -66.093,A -90.000,B 90.000,C 0.000} C_DIS
LIN {X 44.029,Y -45.308,Z -66.420,A -90.000,B 90.000,C 0.000} C_DIS
LIN {X 43.855,Y -45.308,Z -66.723,A -90.000,B 90.000,C 0.000} C_DIS
LIN {X 43.802,Y -45.308,Z -66.798,A -90.000,B 90.000,C 0.000} C_DIS
LIN {X 42.684,Y -45.308,Z -68.268,A -90.000,B 90.000,C 0.000} C_DIS
LIN {X 42.597,Y -45.308,Z -68.377,A -90.000,B 90.000,C 0.000} C_DIS
LIN {X 42.384,Y -45.308,Z -68.615,A -90.000,B 90.000,C 0.000} C_DIS
LIN {X 42.039,Y -45.308,Z -68.934,A -90.000,B 90.000,C 0.000} C_DIS
LIN {X 41.753,Y -45.308,Z -69.138,A -90.000,B 90.000,C 0.000} C_DIS
LIN {X 41.236,Y -45.308,Z -69.483,A -90.000,B 90.000,C 0.000} C_DIS
LIN {X 40.480,Y -45.308,Z -69.899,A -90.000,B 90.000,C 0.000} C_DIS
LIN {X 40.183,Y -45.308,Z -70.015,A -90.000,B 90.000,C 0.000} C_DIS
LIN {X 39.842,Y -45.308,Z -70.114,A -90.000,B 90.000,C 0.000} C_DIS
LIN {X 38.931,Y -45.308,Z -70.395,A -90.000,B 90.000,C 0.000} C_DIS
LIN {X 38.700,Y -45.308,Z -70.446,A -90.000,B 90.000,C 0.000} C_DIS
LIN {X 38.628,Y -45.308,Z -70.458,A -90.000,B 90.000,C 0.000} C_DIS
LIN {X 38.392,Y -45.308,Z -70.472,A -90.000,B 90.000,C 0.000} C_DIS
LIN {X 38.318,Y -45.308,Z -70.470,A -90.000,B 90.000,C 0.000} C_DIS
LIN {X 38.083,Y -45.308,Z -70.447,A -90.000,B 90.000,C 0.000} C_DIS
LIN {X 37.356,Y -45.308,Z -70.340,A -90.000,B 90.000,C 0.000} C_DIS
LIN {X 37.207,Y -45.308,Z -70.316,A -90.000,B 90.000,C 0.000} C_DIS
LIN {X 36.934,Y -45.308,Z -70.245,A -90.000,B 90.000,C 0.000} C_DIS
LIN {X 36.645,Y -45.308,Z -70.121,A -90.000,B 90.000,C 0.000} C_DIS
LIN {X 36.379,Y -45.308,Z -69.952,A -90.000,B 90.000,C 0.000} C_DIS
LIN {X 35.795,Y -45.308,Z -69.573,A -90.000,B 90.000,C 0.000} C_DIS
LIN {X 35.574,Y -45.308,Z -69.376,A -90.000,B 90.000,C 0.000} C_DIS
LIN {X 35.497,Y -45.308,Z -69.284,A -90.000,B 90.000,C 0.000} C_DIS
LIN {X 35.388,Y -45.308,Z -69.146,A -90.000,B 90.000,C 0.000} C_DIS
LIN {X 35.327,Y -45.308,Z -69.042,A -90.000,B 90.000,C 0.000} C_DIS
LIN {X 35.244,Y -45.308,Z -68.887,A -90.000,B 90.000,C 0.000} C_DIS
LIN {X 35.159,Y -45.308,Z -68.695,A -90.000,B 90.000,C 0.000} C_DIS
LIN {X 35.072,Y -45.308,Z -68.427,A -90.000,B 90.000,C 0.000} C_DIS
LIN {X 34.901,Y -45.308,Z -67.813,A -90.000,B 90.000,C 0.000} C_DIS
LIN {X 34.743,Y -45.308,Z -66.978,A -90.000,B 90.000,C 0.000} C_DIS
LIN {X 34.726,Y -45.308,Z -66.719,A -90.000,B 90.000,C 0.000} C_DIS
LIN {X 34.709,Y -45.308,Z -66.365,A -90.000,B 90.000,C 0.000} C_DIS
LIN {X 34.739,Y -45.308,Z -66.037,A -90.000,B 90.000,C 0.000} C_DIS
LIN {X 34.762,Y -45.308,Z -65.933,A -90.000,B 90.000,C 0.000} C_DIS
LIN {X 35.211,Y -45.308,Z -64.131,A -90.000,B 90.000,C 0.000} C_DIS
LIN {X 35.281,Y -45.308,Z -63.948,A -90.000,B 90.000,C 0.000} C_DIS
LIN {X 35.337,Y -45.308,Z -63.818,A -90.000,B 90.000,C 0.000} C_DIS
LIN {X 35.748,Y -45.308,Z -63.072,A -90.000,B 90.000,C 0.000} C_DIS
LIN {X 36.021,Y -45.308,Z -62.613,A -90.000,B 90.000,C 0.000} C_DIS
LIN {X 36.217,Y -45.308,Z -62.239,A -90.000,B 90.000,C 0.000} C_DIS
LIN {X 36.459,Y -45.308,Z -61.838,A -90.000,B 90.000,C 0.000} C_DIS
LIN {X 36.661,Y -45.308,Z -61.573,A -90.000,B 90.000,C 0.000} C_DIS
LIN {X 36.721,Y -45.308,Z -61.499,A -90.000,B 90.000,C 0.000} C_DIS
LIN {X 37.216,Y -45.308,Z -60.970,A -90.000,B 90.000,C 0.000} C_DIS
LIN {X 37.461,Y -45.308,Z -60.765,A -90.000,B 90.000,C 0.000} C_DIS
LIN {X 37.734,Y -45.308,Z -60.549,A -90.000,B 90.000,C 0.000} C_DIS
LIN {X 38.248,Y -45.308,Z -60.092,A -90.000,B 90.000,C 0.000} C_DIS
LIN {X 38.493,Y -45.308,Z -59.886,A -90.000,B 90.000,C 0.000} C_DIS
LIN {X 38.630,Y -45.308,Z -59.791,A -90.000,B 90.000,C 0.000} C_DIS
LIN {X 38.813,Y -45.308,Z -59.681,A -90.000,B 90.000,C 0.000} C_DIS
LIN {X 38.897,Y -45.308,Z -59.639,A -90.000,B 90.000,C 0.000} C_DIS
LIN {X 39.094,Y -45.308,Z -59.559,A -90.000,B 90.000,C 0.000} C_DIS
LIN {X 39.615,Y -45.308,Z -59.399,A -90.000,B 90.000,C 0.000} C_DIS
LIN {X 40.074,Y -45.308,Z -59.286,A -90.000,B 90.000,C 0.000} C_DIS
LIN {X 40.204,Y -45.308,Z -59.256,A -90.000,B 90.000,C 0.000} C_DIS
LIN {X 40.389,Y -45.310,Z -59.211,A -90.000,B 90.000,C 0.000} C_DIS
LIN {X 40.695,Y -45.303,Z -59.175,A -90.000,B 90.000,C 0.000} C_DIS
LIN {X 41.016,Y -45.291,Z -59.174,A -90.000,B 90.000,C 0.000} C_DIS
LIN {X 41.147,Y -45.284,Z -59.189,A -90.000,B 90.000,C 0.000} C_DIS
LIN {X 41.408,Y -45.265,Z -59.213,A -90.000,B 90.000,C 0.000} C_DIS
LIN {X 42.301,Y -45.184,Z -59.264,A -90.000,B 90.000,C 0.000} C_DIS
LIN {X 42.514,Y -45.161,Z -59.290,A -90.000,B 90.000,C 0.000} C_DIS
LIN {X 42.769,Y -45.131,Z -59.349,A -90.000,B 90.000,C 0.000} C_DIS
LIN {X 42.979,Y -45.105,Z -59.418,A -90.000,B 90.000,C 0.000} C_DIS
LIN {X 43.171,Y -45.078,Z -59.500,A -90.000,B 90.000,C 0.000} C_DIS
LIN {X 43.350,Y -45.050,Z -59.589,A -90.000,B 90.000,C 0.000} C_DIS
LIN {X 43.612,Y -44.997,Z -59.723,A -90.000,B 90.000,C 0.000} C_DIS
LIN {X 44.064,Y -44.906,Z -59.935,A -90.000,B 90.000,C 0.000} C_DIS
LIN {X 44.239,Y -44.870,Z -60.027,A -90.000,B 90.000,C 0.000} C_DIS
LIN {X 44.500,Y -44.816,Z -60.172,A -90.000,B 90.000,C 0.000} C_DIS
LIN {X 44.667,Y -44.780,Z -60.278,A -90.000,B 90.000,C 0.000} C_DIS
LIN {X 44.829,Y -44.744,Z -60.392,A -90.000,B 90.000,C 0.000} C_DIS
LIN {X 44.984,Y -44.708,Z -60.516,A -90.000,B 90.000,C 0.000} C_DIS
LIN {X 45.133,Y -44.672,Z -60.650,A -90.000,B 90.000,C 0.000} C_DIS
LIN {X 45.206,Y -44.654,Z -60.719,A -90.000,B 90.000,C 0.000} C_DIS
LIN {X 45.368,Y -44.612,Z -60.884,A -90.000,B 90.000,C 0.000} C_DIS
LIN {X 45.479,Y -44.579,Z -61.026,A -90.000,B 90.000,C 0.000} C_DIS
LIN {X 45.669,Y -44.520,Z -61.291,A -90.000,B 90.000,C 0.000} C_DIS
LIN {X 45.733,Y -44.499,Z -61.386,A -90.000,B 90.000,C 0.000} C_DIS
LIN {X 45.855,Y -44.456,Z -61.586,A -90.000,B 90.000,C 0.000} C_DIS
LIN {X 45.974,Y -44.412,Z -61.802,A -90.000,B 90.000,C 0.000} C_DIS
LIN {X 46.031,Y -44.388,Z -61.916,A -90.000,B 90.000,C 0.000} C_DIS
LIN {X 46.086,Y -44.365,Z -62.034,A -90.000,B 90.000,C 0.000} C_DIS
LIN {X 46.189,Y -44.316,Z -62.282,A -90.000,B 90.000,C 0.000} C_DIS
LIN {X 46.203,Y -44.323,Z -62.312,A -90.000,B 90.000,C 0.000} C_DIS
LIN {X 46.246,Y -44.350,Z -62.422,A -90.000,B 90.000,C 0.000} C_DIS
LIN {X 46.319,Y -44.398,Z -62.624,A -90.000,B 90.000,C 0.000} C_DIS
LIN {X 46.348,Y -44.418,Z -62.708,A -90.000,B 90.000,C 0.000} C_DIS
LIN {X 46.380,Y -44.445,Z -62.798,A -90.000,B 90.000,C 0.000} C_DIS
LIN {X 46.399,Y -44.463,Z -62.860,A -90.000,B 90.000,C 0.000} C_DIS
LIN {X 46.416,Y -44.481,Z -62.922,A -90.000,B 90.000,C 0.000} C_DIS
LIN {X 46.436,Y -44.507,Z -63.012,A -90.000,B 90.000,C 0.000} C_DIS
LIN {X 46.486,Y -44.568,Z -63.338,A -90.000,B 90.000,C 0.000} C_DIS
LIN {X 46.500,Y -44.592,Z -63.471,A -90.000,B 90.000,C 0.000} C_DIS
LIN {X 46.505,Y -44.608,Z -63.575,A -90.000,B 90.000,C 0.000} C_DIS
LIN {X 46.501,Y -44.622,Z -63.716,A -90.000,B 90.000,C 0.000} C_DIS
LIN {X 46.479,Y -44.654,Z -64.052,A -90.000,B 90.000,C 0.000} C_DIS
LIN {X 46.460,Y -44.670,Z -64.217,A -90.000,B 90.000,C 0.000} C_DIS
LIN {X 46.220,Y -44.804,Z -65.705,A -90.000,B 90.000,C 0.000} C_DIS
LIN {X 46.204,Y -44.812,Z -65.800,A -90.000,B 90.000,C 0.000} C_DIS
LIN {X 46.167,Y -44.818,Z -66.006,A -90.000,B 90.000,C 0.000} C_DIS
LIN {X 46.134,Y -44.818,Z -66.172,A -90.000,B 90.000,C 0.000} C_DIS
LIN {X 46.094,Y -44.811,Z -66.335,A -90.000,B 90.000,C 0.000} C_DIS
LIN {X 46.058,Y -44.802,Z -66.469,A -90.000,B 90.000,C 0.000} C_DIS
LIN {X 46.031,Y -44.794,Z -66.572,A -90.000,B 90.000,C 0.000} C_DIS
LIN {X 46.007,Y -44.788,Z -66.652,A -90.000,B 90.000,C 0.000} C_DIS
LIN {X 45.972,Y -44.779,Z -66.750,A -90.000,B 90.000,C 0.000} C_DIS
LIN {X 45.788,Y -44.738,Z -67.181,A -90.000,B 90.000,C 0.000} C_DIS
LIN {X 45.719,Y -44.724,Z -67.314,A -90.000,B 90.000,C 0.000} C_DIS
LIN {X 45.503,Y -44.683,Z -67.668,A -90.000,B 90.000,C 0.000} C_DIS
LIN {X 45.322,Y -44.651,Z -67.913,A -90.000,B 90.000,C 0.000} C_DIS
LIN {X 45.300,Y -44.647,Z -67.946,A -90.000,B 90.000,C 0.000} C_DIS
LIN {X 44.978,Y -44.592,Z -68.337,A -90.000,B 90.000,C 0.000} C_DIS
LIN {X 44.879,Y -44.569,Z -68.452,A -90.000,B 90.000,C 0.000} C_DIS
LIN {X 44.520,Y -44.467,Z -68.851,A -90.000,B 90.000,C 0.000} C_DIS
LIN {X 44.486,Y -44.456,Z -68.888,A -90.000,B 90.000,C 0.000} C_DIS
LIN {X 44.374,Y -44.427,Z -69.011,A -90.000,B 90.000,C 0.000} C_DIS
LIN {X 44.045,Y -44.333,Z -69.361,A -90.000,B 90.000,C 0.000} C_DIS
LIN {X 43.950,Y -44.307,Z -69.457,A -90.000,B 90.000,C 0.000} C_DIS
LIN {X 43.857,Y -44.284,Z -69.544,A -90.000,B 90.000,C 0.000} C_DIS
LIN {X 43.654,Y -44.259,Z -69.750,A -90.000,B 90.000,C 0.000} C_DIS
LIN {X 43.563,Y -44.251,Z -69.837,A -90.000,B 90.000,C 0.000} C_DIS
LIN {X 43.183,Y -44.230,Z -70.171,A -90.000,B 90.000,C 0.000} C_DIS
LIN {X 43.018,Y -44.228,Z -70.303,A -90.000,B 90.000,C 0.000} C_DIS
LIN {X 42.735,Y -44.234,Z -70.510,A -90.000,B 90.000,C 0.000} C_DIS
LIN {X 42.180,Y -44.256,Z -70.898,A -90.000,B 90.000,C 0.000} C_DIS
LIN {X 42.116,Y -44.259,Z -70.941,A -90.000,B 90.000,C 0.000} C_DIS
LIN {X 41.790,Y -44.279,Z -71.136,A -90.000,B 90.000,C 0.000} C_DIS
LIN {X 41.551,Y -44.288,Z -71.273,A -90.000,B 90.000,C 0.000} C_DIS
LIN {X 41.308,Y -44.287,Z -71.406,A -90.000,B 90.000,C 0.000} C_DIS
LIN {X 41.224,Y -44.287,Z -71.450,A -90.000,B 90.000,C 0.000} C_DIS
LIN {X 41.106,Y -44.289,Z -71.502,A -90.000,B 90.000,C 0.000} C_DIS
LIN {X 40.810,Y -44.298,Z -71.623,A -90.000,B 90.000,C 0.000} C_DIS
LIN {X 40.662,Y -44.306,Z -71.678,A -90.000,B 90.000,C 0.000} C_DIS
LIN {X 40.342,Y -44.331,Z -71.786,A -90.000,B 90.000,C 0.000} C_DIS
LIN {X 40.151,Y -44.343,Z -71.852,A -90.000,B 90.000,C 0.000} C_DIS
LIN {X 39.395,Y -44.360,Z -72.094,A -90.000,B 90.000,C 0.000} C_DIS
LIN {X 39.332,Y -44.363,Z -72.111,A -90.000,B 90.000,C 0.000} C_DIS
LIN {X 39.028,Y -44.360,Z -72.176,A -90.000,B 90.000,C 0.000} C_DIS
LIN {X 38.979,Y -44.360,Z -72.184,A -90.000,B 90.000,C 0.000} C_DIS
LIN {X 38.882,Y -44.360,Z -72.200,A -90.000,B 90.000,C 0.000} C_DIS
LIN {X 38.700,Y -44.364,Z -72.219,A -90.000,B 90.000,C 0.000} C_DIS
LIN {X 38.453,Y -44.373,Z -72.238,A -90.000,B 90.000,C 0.000} C_DIS
LIN {X 38.292,Y -44.383,Z -72.243,A -90.000,B 90.000,C 0.000} C_DIS
LIN {X 38.231,Y -44.388,Z -72.244,A -90.000,B 90.000,C 0.000} C_DIS
LIN {X 38.011,Y -44.412,Z -72.237,A -90.000,B 90.000,C 0.000} C_DIS
LIN {X 37.817,Y -44.431,Z -72.225,A -90.000,B 90.000,C 0.000} C_DIS
LIN {X 37.736,Y -44.439,Z -72.217,A -90.000,B 90.000,C 0.000} C_DIS
LIN {X 37.468,Y -44.462,Z -72.188,A -90.000,B 90.000,C 0.000} C_DIS
LIN {X 37.089,Y -44.469,Z -72.135,A -90.000,B 90.000,C 0.000} C_DIS
LIN {X 36.847,Y -44.472,Z -72.097,A -90.000,B 90.000,C 0.000} C_DIS
LIN {X 36.750,Y -44.476,Z -72.076,A -90.000,B 90.000,C 0.000} C_DIS
LIN {X 36.423,Y -44.493,Z -71.998,A -90.000,B 90.000,C 0.000} C_DIS
LIN {X 36.341,Y -44.497,Z -71.974,A -90.000,B 90.000,C 0.000} C_DIS
LIN {X 36.191,Y -44.504,Z -71.919,A -90.000,B 90.000,C 0.000} C_DIS
LIN {X 36.071,Y -44.512,Z -71.871,A -90.000,B 90.000,C 0.000} C_DIS
LIN {X 35.881,Y -44.511,Z -71.789,A -90.000,B 90.000,C 0.000} C_DIS
LIN {X 35.780,Y -44.514,Z -71.739,A -90.000,B 90.000,C 0.000} C_DIS
LIN {X 35.651,Y -44.516,Z -71.665,A -90.000,B 90.000,C 0.000} C_DIS
LIN {X 35.270,Y -44.530,Z -71.429,A -90.000,B 90.000,C 0.000} C_DIS
LIN {X 34.917,Y -44.531,Z -71.200,A -90.000,B 90.000,C 0.000} C_DIS
LIN {X 34.728,Y -44.519,Z -71.069,A -90.000,B 90.000,C 0.000} C_DIS
LIN {X 34.663,Y -44.517,Z -71.019,A -90.000,B 90.000,C 0.000} C_DIS
LIN {X 34.548,Y -44.507,Z -70.915,A -90.000,B 90.000,C 0.000} C_DIS
LIN {X 34.439,Y -44.498,Z -70.814,A -90.000,B 90.000,C 0.000} C_DIS
LIN {X 34.365,Y -44.489,Z -70.743,A -90.000,B 90.000,C 0.000} C_DIS
LIN {X 34.274,Y -44.481,Z -70.651,A -90.000,B 90.000,C 0.000} C_DIS
LIN {X 34.207,Y -44.476,Z -70.576,A -90.000,B 90.000,C 0.000} C_DIS
LIN {X 34.072,Y -44.470,Z -70.409,A -90.000,B 90.000,C 0.000} C_DIS
LIN {X 33.966,Y -44.461,Z -70.269,A -90.000,B 90.000,C 0.000} C_DIS
LIN {X 33.902,Y -44.457,Z -70.178,A -90.000,B 90.000,C 0.000} C_DIS
LIN {X 33.849,Y -44.455,Z -70.097,A -90.000,B 90.000,C 0.000} C_DIS
LIN {X 33.774,Y -44.446,Z -69.962,A -90.000,B 90.000,C 0.000} C_DIS
LIN {X 33.641,Y -44.435,Z -69.705,A -90.000,B 90.000,C 0.000} C_DIS
LIN {X 33.578,Y -44.428,Z -69.560,A -90.000,B 90.000,C 0.000} C_DIS
LIN {X 33.511,Y -44.423,Z -69.401,A -90.000,B 90.000,C 0.000} C_DIS
LIN {X 33.467,Y -44.412,Z -69.270,A -90.000,B 90.000,C 0.000} C_DIS
LIN {X 33.433,Y -44.405,Z -69.155,A -90.000,B 90.000,C 0.000} C_DIS
LIN {X 33.361,Y -44.390,Z -68.904,A -90.000,B 90.000,C 0.000} C_DIS
LIN {X 33.269,Y -44.376,Z -68.548,A -90.000,B 90.000,C 0.000} C_DIS
LIN {X 33.205,Y -44.360,Z -68.286,A -90.000,B 90.000,C 0.000} C_DIS
LIN {X 33.186,Y -44.356,Z -68.204,A -90.000,B 90.000,C 0.000} C_DIS
LIN {X 33.160,Y -44.350,Z -68.054,A -90.000,B 90.000,C 0.000} C_DIS
LIN {X 33.102,Y -44.331,Z -67.692,A -90.000,B 90.000,C 0.000} C_DIS
LIN {X 33.054,Y -44.285,Z -67.297,A -90.000,B 90.000,C 0.000} C_DIS
LIN {X 33.049,Y -44.279,Z -67.241,A -90.000,B 90.000,C 0.000} C_DIS
LIN {X 33.044,Y -44.259,Z -67.087,A -90.000,B 90.000,C 0.000} C_DIS
LIN {X 33.045,Y -44.225,Z -66.754,A -90.000,B 90.000,C 0.000} C_DIS
LIN {X 33.049,Y -44.196,Z -66.444,A -90.000,B 90.000,C 0.000} C_DIS
LIN {X 33.054,Y -44.187,Z -66.316,A -90.000,B 90.000,C 0.000} C_DIS
LIN {X 33.062,Y -44.183,Z -66.219,A -90.000,B 90.000,C 0.000} C_DIS
LIN {X 33.096,Y -44.177,Z -65.887,A -90.000,B 90.000,C 0.000} C_DIS
LIN {X 33.111,Y -44.175,Z -65.777,A -90.000,B 90.000,C 0.000} C_DIS
LIN {X 33.132,Y -44.176,Z -65.668,A -90.000,B 90.000,C 0.000} C_DIS
LIN {X 33.220,Y -44.179,Z -65.296,A -90.000,B 90.000,C 0.000} C_DIS
LIN {X 33.608,Y -44.153,Z -63.812,A -90.000,B 90.000,C 0.000} C_DIS
LIN {X 33.630,Y -44.148,Z -63.738,A -90.000,B 90.000,C 0.000} C_DIS
LIN {X 33.665,Y -44.143,Z -63.628,A -90.000,B 90.000,C 0.000} C_DIS
LIN {X 33.737,Y -44.144,Z -63.432,A -90.000,B 90.000,C 0.000} C_DIS
LIN {X 33.812,Y -44.147,Z -63.243,A -90.000,B 90.000,C 0.000} C_DIS
LIN {X 33.843,Y -44.149,Z -63.167,A -90.000,B 90.000,C 0.000} C_DIS
LIN {X 33.907,Y -44.153,Z -63.029,A -90.000,B 90.000,C 0.000} C_DIS
LIN {X 34.316,Y -44.203,Z -62.219,A -90.000,B 90.000,C 0.000} C_DIS
LIN {X 34.409,Y -44.216,Z -62.045,A -90.000,B 90.000,C 0.000} C_DIS
LIN {X 34.562,Y -44.230,Z -61.767,A -90.000,B 90.000,C 0.000} C_DIS
LIN {X 34.732,Y -44.217,Z -61.460,A -90.000,B 90.000,C 0.000} C_DIS
LIN {X 34.782,Y -44.215,Z -61.374,A -90.000,B 90.000,C 0.000} C_DIS
LIN {X 35.026,Y -44.212,Z -60.974,A -90.000,B 90.000,C 0.000} C_DIS
LIN {X 35.128,Y -44.216,Z -60.819,A -90.000,B 90.000,C 0.000} C_DIS
LIN {X 35.355,Y -44.236,Z -60.503,A -90.000,B 90.000,C 0.000} C_DIS
LIN {X 35.430,Y -44.243,Z -60.404,A -90.000,B 90.000,C 0.000} C_DIS
LIN {X 35.539,Y -44.258,Z -60.271,A -90.000,B 90.000,C 0.000} C_DIS
LIN {X 35.784,Y -44.282,Z -59.988,A -90.000,B 90.000,C 0.000} C_DIS
LIN {X 35.973,Y -44.296,Z -59.775,A -90.000,B 90.000,C 0.000} C_DIS
LIN {X 36.018,Y -44.298,Z -59.728,A -90.000,B 90.000,C 0.000} C_DIS
LIN {X 36.125,Y -44.303,Z -59.628,A -90.000,B 90.000,C 0.000} C_DIS
LIN {X 36.383,Y -44.320,Z -59.400,A -90.000,B 90.000,C 0.000} C_DIS
LIN {X 36.610,Y -44.338,Z -59.209,A -90.000,B 90.000,C 0.000} C_DIS
LIN {X 37.128,Y -44.356,Z -58.736,A -90.000,B 90.000,C 0.000} C_DIS
LIN {X 37.411,Y -44.346,Z -58.507,A -90.000,B 90.000,C 0.000} C_DIS
LIN {X 37.631,Y -44.340,Z -58.354,A -90.000,B 90.000,C 0.000} C_DIS
LIN {X 37.697,Y -44.340,Z -58.311,A -90.000,B 90.000,C 0.000} C_DIS
LIN {X 37.911,Y -44.343,Z -58.180,A -90.000,B 90.000,C 0.000} C_DIS
LIN {X 37.998,Y -44.346,Z -58.128,A -90.000,B 90.000,C 0.000} C_DIS
LIN {X 38.106,Y -44.352,Z -58.070,A -90.000,B 90.000,C 0.000} C_DIS
LIN {X 38.210,Y -44.360,Z -58.017,A -90.000,B 90.000,C 0.000} C_DIS
LIN {X 38.329,Y -44.371,Z -57.962,A -90.000,B 90.000,C 0.000} C_DIS
LIN {X 38.444,Y -44.377,Z -57.913,A -90.000,B 90.000,C 0.000} C_DIS
LIN {X 38.590,Y -44.388,Z -57.857,A -90.000,B 90.000,C 0.000} C_DIS
LIN {X 38.718,Y -44.398,Z -57.812,A -90.000,B 90.000,C 0.000} C_DIS
LIN {X 39.015,Y -44.409,Z -57.715,A -90.000,B 90.000,C 0.000} C_DIS
LIN {X 39.164,Y -44.406,Z -57.673,A -90.000,B 90.000,C 0.000} C_DIS
LIN {X 39.188,Y -44.406,Z -57.666,A -90.000,B 90.000,C 0.000} C_DIS
LIN {X 39.670,Y -44.408,Z -57.547,A -90.000,B 90.000,C 0.000} C_DIS
LIN {X 40.033,Y -44.412,Z -57.462,A -90.000,B 90.000,C 0.000} C_DIS
LIN {X 40.184,Y -44.416,Z -57.436,A -90.000,B 90.000,C 0.000} C_DIS
LIN {X 40.306,Y -44.423,Z -57.422,A -90.000,B 90.000,C 0.000} C_DIS
LIN {X 40.625,Y -44.423,Z -57.399,A -90.000,B 90.000,C 0.000} C_DIS
LIN {X 40.730,Y -44.419,Z -57.400,A -90.000,B 90.000,C 0.000} C_DIS
LIN {X 40.855,Y -44.418,Z -57.407,A -90.000,B 90.000,C 0.000} C_DIS
LIN {X 40.943,Y -44.418,Z -57.414,A -90.000,B 90.000,C 0.000} C_DIS
LIN {X 41.173,Y -44.405,Z -57.440,A -90.000,B 90.000,C 0.000} C_DIS
LIN {X 41.433,Y -44.400,Z -57.485,A -90.000,B 90.000,C 0.000} C_DIS
LIN {X 42.007,Y -44.405,Z -57.618,A -90.000,B 90.000,C 0.000} C_DIS
LIN {X 42.264,Y -44.405,Z -57.681,A -90.000,B 90.000,C 0.000} C_DIS
LIN {X 42.399,Y -44.397,Z -57.721,A -90.000,B 90.000,C 0.000} C_DIS
LIN {X 42.677,Y -44.383,Z -57.808,A -90.000,B 90.000,C 0.000} C_DIS
LIN {X 42.791,Y -44.372,Z -57.848,A -90.000,B 90.000,C 0.000} C_DIS
LIN {X 42.983,Y -44.357,Z -57.923,A -90.000,B 90.000,C 0.000} C_DIS
LIN {X 43.268,Y -44.320,Z -58.067,A -90.000,B 90.000,C 0.000} C_DIS
LIN {X 43.390,Y -44.306,Z -58.134,A -90.000,B 90.000,C 0.000} C_DIS
LIN {X 43.513,Y -44.296,Z -58.212,A -90.000,B 90.000,C 0.000} C_DIS
LIN {X 43.758,Y -44.281,Z -58.375,A -90.000,B 90.000,C 0.000} C_DIS
LIN {X 43.813,Y -44.278,Z -58.414,A -90.000,B 90.000,C 0.000} C_DIS
LIN {X 43.918,Y -44.272,Z -58.496,A -90.000,B 90.000,C 0.000} C_DIS
LIN {X 44.183,Y -44.268,Z -58.726,A -90.000,B 90.000,C 0.000} C_DIS
LIN {X 44.277,Y -44.270,Z -58.815,A -90.000,B 90.000,C 0.000} C_DIS
LIN {X 44.319,Y -44.270,Z -58.858,A -90.000,B 90.000,C 0.000} C_DIS
LIN {X 44.388,Y -44.274,Z -58.931,A -90.000,B 90.000,C 0.000} C_DIS
LIN {X 44.601,Y -44.290,Z -59.170,A -90.000,B 90.000,C 0.000} C_DIS
LIN {X 44.657,Y -44.297,Z -59.238,A -90.000,B 90.000,C 0.000} C_DIS
LIN {X 44.726,Y -44.304,Z -59.326,A -90.000,B 90.000,C 0.000} C_DIS
LIN {X 44.809,Y -44.314,Z -59.441,A -90.000,B 90.000,C 0.000} C_DIS
LIN {X 44.949,Y -44.336,Z -59.646,A -90.000,B 90.000,C 0.000} C_DIS
LIN {X 45.021,Y -44.344,Z -59.757,A -90.000,B 90.000,C 0.000} C_DIS
LIN {X 45.302,Y -44.366,Z -60.232,A -90.000,B 90.000,C 0.000} C_DIS
LIN {X 45.474,Y -44.364,Z -60.542,A -90.000,B 90.000,C 0.000} C_DIS
LIN {X 45.532,Y -44.358,Z -60.666,A -90.000,B 90.000,C 0.000} C_DIS
LIN {X 45.768,Y -44.335,Z -61.208,A -90.000,B 90.000,C 0.000} C_DIS
LIN {X 45.853,Y -44.320,Z -61.416,A -90.000,B 90.000,C 0.000} C_DIS
LIN {X 46.044,Y -44.310,Z -61.901,A -90.000,B 90.000,C 0.000} C_DIS
LIN {X 46.093,Y -44.307,Z -62.032,A -90.000,B 90.000,C 0.000} C_DIS
LIN {X 46.166,Y -44.304,Z -62.232,A -90.000,B 90.000,C 0.000} C_DIS
LIN {X 46.189,Y -44.316,Z -62.282,A -90.000,B 90.000,C 0.000} C_DIS
LIN {X 46.418,Y -43.924,Z -60.722,A -90.000,B 90.000,C 0.000} C_DIS
LIN {X 46.503,Y -43.742,Z -60.149,A -90.000,B 90.000,C 0.000} C_DIS
LIN {X 46.576,Y -43.526,Z -59.650,A -90.000,B 90.000,C 0.000} C_DIS
LIN {X 46.648,Y -43.308,Z -59.163,A -90.000,B 90.000,C 0.000} C_DIS
LIN {X 46.752,Y -43.360,Z -59.286,A -90.000,B 90.000,C 0.000} C_DIS
LIN {X 46.939,Y -43.466,Z -59.500,A -90.000,B 90.000,C 0.000} C_DIS
LIN {X 47.097,Y -43.561,Z -59.693,A -90.000,B 90.000,C 0.000} C_DIS
LIN {X 47.229,Y -43.651,Z -59.878,A -90.000,B 90.000,C 0.000} C_DIS
LIN {X 47.341,Y -43.731,Z -60.057,A -90.000,B 90.000,C 0.000} C_DIS
LIN {X 47.499,Y -43.851,Z -60.325,A -90.000,B 90.000,C 0.000} C_DIS
LIN {X 47.513,Y -43.862,Z -60.349,A -90.000,B 90.000,C 0.000} C_DIS
LIN {X 47.611,Y -43.924,Z -60.539,A -90.000,B 90.000,C 0.000} C_DIS
LIN {X 47.666,Y -43.960,Z -60.651,A -90.000,B 90.000,C 0.000} C_DIS
LIN {X 47.785,Y -44.043,Z -60.916,A -90.000,B 90.000,C 0.000} C_DIS
LIN {X 47.904,Y -44.124,Z -61.192,A -90.000,B 90.000,C 0.000} C_DIS
LIN {X 47.969,Y -44.169,Z -61.352,A -90.000,B 90.000,C 0.000} C_DIS
LIN {X 48.024,Y -44.206,Z -61.493,A -90.000,B 90.000,C 0.000} C_DIS
LIN {X 48.068,Y -44.233,Z -61.596,A -90.000,B 90.000,C 0.000} C_DIS
LIN {X 48.131,Y -44.276,Z -61.757,A -90.000,B 90.000,C 0.000} C_DIS
LIN {X 48.268,Y -44.378,Z -62.142,A -90.000,B 90.000,C 0.000} C_DIS
LIN {X 48.306,Y -44.409,Z -62.257,A -90.000,B 90.000,C 0.000} C_DIS
LIN {X 48.341,Y -44.442,Z -62.379,A -90.000,B 90.000,C 0.000} C_DIS
LIN {X 48.374,Y -44.478,Z -62.512,A -90.000,B 90.000,C 0.000} C_DIS
LIN {X 48.400,Y -44.510,Z -62.632,A -90.000,B 90.000,C 0.000} C_DIS
LIN {X 48.435,Y -44.570,Z -62.853,A -90.000,B 90.000,C 0.000} C_DIS
LIN {X 48.461,Y -44.617,Z -63.030,A -90.000,B 90.000,C 0.000} C_DIS
LIN {X 48.476,Y -44.652,Z -63.159,A -90.000,B 90.000,C 0.000} C_DIS
LIN {X 48.488,Y -44.673,Z -63.267,A -90.000,B 90.000,C 0.000} C_DIS
LIN {X 48.494,Y -44.691,Z -63.363,A -90.000,B 90.000,C 0.000} C_DIS
LIN {X 48.501,Y -44.725,Z -63.543,A -90.000,B 90.000,C 0.000} C_DIS
LIN {X 48.498,Y -44.750,Z -63.693,A -90.000,B 90.000,C 0.000} C_DIS
LIN {X 48.494,Y -44.762,Z -63.817,A -90.000,B 90.000,C 0.000} C_DIS
LIN {X 48.471,Y -44.793,Z -64.163,A -90.000,B 90.000,C 0.000} C_DIS
LIN {X 48.453,Y -44.810,Z -64.345,A -90.000,B 90.000,C 0.000} C_DIS
LIN {X 48.444,Y -44.818,Z -64.427,A -90.000,B 90.000,C 0.000} C_DIS
LIN {X 48.347,Y -44.875,Z -65.041,A -90.000,B 90.000,C 0.000} C_DIS
LIN {X 48.219,Y -44.948,Z -65.832,A -90.000,B 90.000,C 0.000} C_DIS
LIN {X 48.188,Y -44.962,Z -66.024,A -90.000,B 90.000,C 0.000} C_DIS
LIN {X 48.130,Y -44.977,Z -66.354,A -90.000,B 90.000,C 0.000} C_DIS
LIN {X 48.113,Y -44.976,Z -66.440,A -90.000,B 90.000,C 0.000} C_DIS
LIN {X 48.087,Y -44.969,Z -66.576,A -90.000,B 90.000,C 0.000} C_DIS
LIN {X 48.056,Y -44.962,Z -66.712,A -90.000,B 90.000,C 0.000} C_DIS
LIN {X 47.960,Y -44.935,Z -67.083,A -90.000,B 90.000,C 0.000} C_DIS
LIN {X 47.915,Y -44.923,Z -67.237,A -90.000,B 90.000,C 0.000} C_DIS
LIN {X 47.867,Y -44.911,Z -67.378,A -90.000,B 90.000,C 0.000} C_DIS
LIN {X 47.832,Y -44.903,Z -67.475,A -90.000,B 90.000,C 0.000} C_DIS
LIN {X 47.620,Y -44.860,Z -67.975,A -90.000,B 90.000,C 0.000} C_DIS
LIN {X 47.550,Y -44.846,Z -68.122,A -90.000,B 90.000,C 0.000} C_DIS
LIN {X 47.472,Y -44.832,Z -68.272,A -90.000,B 90.000,C 0.000} C_DIS
LIN {X 47.418,Y -44.823,Z -68.366,A -90.000,B 90.000,C 0.000} C_DIS
LIN {X 47.189,Y -44.784,Z -68.739,A -90.000,B 90.000,C 0.000} C_DIS
LIN {X 47.142,Y -44.775,Z -68.810,A -90.000,B 90.000,C 0.000} C_DIS
LIN {X 47.092,Y -44.762,Z -68.881,A -90.000,B 90.000,C 0.000} C_DIS
LIN {X 46.961,Y -44.720,Z -69.058,A -90.000,B 90.000,C 0.000} C_DIS
LIN {X 46.908,Y -44.703,Z -69.134,A -90.000,B 90.000,C 0.000} C_DIS
LIN {X 46.847,Y -44.684,Z -69.213,A -90.000,B 90.000,C 0.000} C_DIS
LIN {X 46.777,Y -44.663,Z -69.299,A -90.000,B 90.000,C 0.000} C_DIS
LIN {X 46.498,Y -44.569,Z -69.636,A -90.000,B 90.000,C 0.000} C_DIS
LIN {X 46.371,Y -44.527,Z -69.783,A -90.000,B 90.000,C 0.000} C_DIS
LIN {X 45.866,Y -44.368,Z -70.342,A -90.000,B 90.000,C 0.000} C_DIS
LIN {X 45.470,Y -44.246,Z -70.762,A -90.000,B 90.000,C 0.000} C_DIS
LIN {X 45.328,Y -44.204,Z -70.903,A -90.000,B 90.000,C 0.000} C_DIS
LIN {X 45.227,Y -44.175,Z -70.999,A -90.000,B 90.000,C 0.000} C_DIS
LIN {X 45.042,Y -44.104,Z -71.181,A -90.000,B 90.000,C 0.000} C_DIS
LIN {X 44.948,Y -44.069,Z -71.268,A -90.000,B 90.000,C 0.000} C_DIS
LIN {X 44.795,Y -44.015,Z -71.399,A -90.000,B 90.000,C 0.000} C_DIS
LIN {X 44.522,Y -43.913,Z -71.622,A -90.000,B 90.000,C 0.000} C_DIS
LIN {X 44.417,Y -43.873,Z -71.704,A -90.000,B 90.000,C 0.000} C_DIS
LIN {X 44.245,Y -43.813,Z -71.827,A -90.000,B 90.000,C 0.000} C_DIS
LIN {X 44.169,Y -43.787,Z -71.878,A -90.000,B 90.000,C 0.000} C_DIS
LIN {X 43.820,Y -43.673,Z -72.094,A -90.000,B 90.000,C 0.000} C_DIS
LIN {X 43.636,Y -43.615,Z -72.198,A -90.000,B 90.000,C 0.000} C_DIS
LIN {X 43.422,Y -43.552,Z -72.318,A -90.000,B 90.000,C 0.000} C_DIS
LIN {X 43.164,Y -43.478,Z -72.456,A -90.000,B 90.000,C 0.000} C_DIS
LIN {X 43.014,Y -43.438,Z -72.528,A -90.000,B 90.000,C 0.000} C_DIS
LIN {X 42.858,Y -43.398,Z -72.595,A -90.000,B 90.000,C 0.000} C_DIS
LIN {X 42.624,Y -43.348,Z -72.697,A -90.000,B 90.000,C 0.000} C_DIS
LIN {X 42.436,Y -43.308,Z -72.776,A -90.000,B 90.000,C 0.000} C_DIS
LIN {X 42.436,Y -60.000,Z -72.776,A -90.000,B 90.000,C 0.000} C_DIS
LIN {X 48.978,Y -60.000,Z -58.970,A -90.000,B 90.000,C 0.000} C_DIS
LIN {X 48.978,Y -43.308,Z -58.970,A -90.000,B 90.000,C 0.000} C_DIS
LIN {X 49.092,Y -43.388,Z -59.154,A -90.000,B 90.000,C 0.000} C_DIS
LIN {X 49.264,Y -43.516,Z -59.447,A -90.000,B 90.000,C 0.000} C_DIS
LIN {X 49.309,Y -43.550,Z -59.527,A -90.000,B 90.000,C 0.000} C_DIS
LIN {X 49.466,Y -43.680,Z -59.826,A -90.000,B 90.000,C 0.000} C_DIS
LIN {X 49.556,Y -43.762,Z -60.015,A -90.000,B 90.000,C 0.000} C_DIS
LIN {X 49.612,Y -43.811,Z -60.134,A -90.000,B 90.000,C 0.000} C_DIS
LIN {X 49.767,Y -43.951,Z -60.485,A -90.000,B 90.000,C 0.000} C_DIS
LIN {X 49.842,Y -44.004,Z -60.671,A -90.000,B 90.000,C 0.000} C_DIS
LIN {X 49.884,Y -44.033,Z -60.778,A -90.000,B 90.000,C 0.000} C_DIS
LIN {X 49.938,Y -44.067,Z -60.908,A -90.000,B 90.000,C 0.000} C_DIS
LIN {X 49.976,Y -44.091,Z -61.003,A -90.000,B 90.000,C 0.000} C_DIS
LIN {X 50.042,Y -44.126,Z -61.182,A -90.000,B 90.000,C 0.000} C_DIS
LIN {X 50.110,Y -44.166,Z -61.375,A -90.000,B 90.000,C 0.000} C_DIS
LIN {X 50.179,Y -44.203,Z -61.578,A -90.000,B 90.000,C 0.000} C_DIS
LIN {X 50.233,Y -44.236,Z -61.751,A -90.000,B 90.000,C 0.000} C_DIS
LIN {X 50.286,Y -44.273,Z -61.945,A -90.000,B 90.000,C 0.000} C_DIS
LIN {X 50.331,Y -44.311,Z -62.135,A -90.000,B 90.000,C 0.000} C_DIS
LIN {X 50.357,Y -44.336,Z -62.260,A -90.000,B 90.000,C 0.000} C_DIS
LIN {X 50.375,Y -44.357,Z -62.360,A -90.000,B 90.000,C 0.000} C_DIS
LIN {X 50.432,Y -44.438,Z -62.741,A -90.000,B 90.000,C 0.000} C_DIS
LIN {X 50.447,Y -44.461,Z -62.845,A -90.000,B 90.000,C 0.000} C_DIS
LIN {X 50.472,Y -44.512,Z -63.073,A -90.000,B 90.000,C 0.000} C_DIS
LIN {X 50.486,Y -44.553,Z -63.250,A -90.000,B 90.000,C 0.000} C_DIS
LIN {X 50.498,Y -44.615,Z -63.517,A -90.000,B 90.000,C 0.000} C_DIS
LIN {X 50.497,Y -44.632,Z -63.618,A -90.000,B 90.000,C 0.000} C_DIS
LIN {X 50.491,Y -44.668,Z -63.855,A -90.000,B 90.000,C 0.000} C_DIS
LIN {X 50.482,Y -44.696,Z -64.037,A -90.000,B 90.000,C 0.000} C_DIS
LIN {X 50.475,Y -44.707,Z -64.151,A -90.000,B 90.000,C 0.000} C_DIS
LIN {X 50.459,Y -44.721,Z -64.367,A -90.000,B 90.000,C 0.000} C_DIS
LIN {X 50.436,Y -44.736,Z -64.595,A -90.000,B 90.000,C 0.000} C_DIS
LIN {X 50.417,Y -44.747,Z -64.747,A -90.000,B 90.000,C 0.000} C_DIS
LIN {X 50.365,Y -44.770,Z -65.074,A -90.000,B 90.000,C 0.000} C_DIS
LIN {X 50.169,Y -44.875,Z -66.293,A -90.000,B 90.000,C 0.000} C_DIS
LIN {X 50.099,Y -44.892,Z -66.691,A -90.000,B 90.000,C 0.000} C_DIS
LIN {X 50.072,Y -44.889,Z -66.837,A -90.000,B 90.000,C 0.000} C_DIS
LIN {X 50.034,Y -44.881,Z -67.027,A -90.000,B 90.000,C 0.000} C_DIS
LIN {X 49.991,Y -44.871,Z -67.206,A -90.000,B 90.000,C 0.000} C_DIS
LIN {X 49.873,Y -44.829,Z -67.655,A -90.000,B 90.000,C 0.000} C_DIS
LIN {X 49.809,Y -44.812,Z -67.869,A -90.000,B 90.000,C 0.000} C_DIS
LIN {X 49.747,Y -44.799,Z -68.051,A -90.000,B 90.000,C 0.000} C_DIS
LIN {X 49.712,Y -44.792,Z -68.148,A -90.000,B 90.000,C 0.000} C_DIS
LIN {X 49.674,Y -44.785,Z -68.245,A -90.000,B 90.000,C 0.000} C_DIS
LIN {X 49.457,Y -44.750,Z -68.758,A -90.000,B 90.000,C 0.000} C_DIS
LIN {X 49.346,Y -44.734,Z -68.994,A -90.000,B 90.000,C 0.000} C_DIS
LIN {X 49.233,Y -44.719,Z -69.214,A -90.000,B 90.000,C 0.000} C_DIS
LIN {X 49.163,Y -44.698,Z -69.334,A -90.000,B 90.000,C 0.000} C_DIS
LIN {X 48.963,Y -44.643,Z -69.661,A -90.000,B 90.000,C 0.000} C_DIS
LIN {X 48.871,Y -44.608,Z -69.806,A -90.000,B 90.000,C 0.000} C_DIS
LIN {X 48.776,Y -44.575,Z -69.946,A -90.000,B 90.000,C 0.000} C_DIS
LIN {X 48.577,Y -44.510,Z -70.220,A -90.000,B 90.000,C 0.000} C_DIS
LIN {X 48.508,Y -44.487,Z -70.316,A -90.000,B 90.000,C 0.000} C_DIS
LIN {X 48.408,Y -44.457,Z -70.443,A -90.000,B 90.000,C 0.000} C_DIS
LIN {X 48.032,Y -44.353,Z -70.901,A -90.000,B 90.000,C 0.000} C_DIS
LIN {X 47.876,Y -44.311,Z -71.082,A -90.000,B 90.000,C 0.000} C_DIS
LIN {X 47.582,Y -44.237,Z -71.411,A -90.000,B 90.000,C 0.000} C_DIS
LIN {X 47.343,Y -44.157,Z -71.674,A -90.000,B 90.000,C 0.000} C_DIS
LIN {X 47.197,Y -44.109,Z -71.829,A -90.000,B 90.000,C 0.000} C_DIS
LIN {X 46.903,Y -43.994,Z -72.135,A -90.000,B 90.000,C 0.000} C_DIS
LIN {X 46.671,Y -43.908,Z -72.358,A -90.000,B 90.000,C 0.000} C_DIS
LIN {X 46.482,Y -43.837,Z -72.543,A -90.000,B 90.000,C 0.000} C_DIS
LIN {X 46.293,Y -43.771,Z -72.718,A -90.000,B 90.000,C 0.000} C_DIS
LIN {X 46.072,Y -43.694,Z -72.905,A -90.000,B 90.000,C 0.000} C_DIS
LIN {X 45.802,Y -43.601,Z -73.127,A -90.000,B 90.000,C 0.000} C_DIS
LIN {X 45.652,Y -43.550,Z -73.243,A -90.000,B 90.000,C 0.000} C_DIS
LIN {X 45.424,Y -43.472,Z -73.406,A -90.000,B 90.000,C 0.000} C_DIS
LIN {X 45.287,Y -43.423,Z -73.496,A -90.000,B 90.000,C 0.000} C_DIS
LIN {X 44.952,Y -43.308,Z -73.702,A -90.000,B 90.000,C 0.000} C_DIS
LIN {X 44.952,Y -60.000,Z -73.702,A -90.000,B 90.000,C 0.000} C_DIS
LIN {X 51.456,Y -60.000,Z -59.545,A -90.000,B 90.000,C 0.000} C_DIS
LIN {X 51.456,Y -43.308,Z -59.545,A -90.000,B 90.000,C 0.000} C_DIS
LIN {X 51.688,Y -43.495,Z -60.093,A -90.000,B 90.000,C 0.000} C_DIS
LIN {X 51.752,Y -43.547,Z -60.244,A -90.000,B 90.000,C 0.000} C_DIS
LIN {X 51.826,Y -43.606,Z -60.418,A -90.000,B 90.000,C 0.000} C_DIS
LIN {X 51.865,Y -43.639,Z -60.514,A -90.000,B 90.000,C 0.000} C_DIS
LIN {X 52.014,Y -43.761,Z -60.908,A -90.000,B 90.000,C 0.000} C_DIS
LIN {X 52.071,Y -43.802,Z -61.068,A -90.000,B 90.000,C 0.000} C_DIS
LIN {X 52.143,Y -43.847,Z -61.305,A -90.000,B 90.000,C 0.000} C_DIS
LIN {X 52.211,Y -43.891,Z -61.563,A -90.000,B 90.000,C 0.000} C_DIS
LIN {X 52.267,Y -43.933,Z -61.807,A -90.000,B 90.000,C 0.000} C_DIS
LIN {X 52.303,Y -43.964,Z -61.986,A -90.000,B 90.000,C 0.000} C_DIS
LIN {X 52.329,Y -43.990,Z -62.145,A -90.000,B 90.000,C 0.000} C_DIS
LIN {X 52.393,Y -44.066,Z -62.606,A -90.000,B 90.000,C 0.000} C_DIS
LIN {X 52.429,Y -44.119,Z -62.946,A -90.000,B 90.000,C 0.000} C_DIS
LIN {X 52.446,Y -44.158,Z -63.178,A -90.000,B 90.000,C 0.000} C_DIS
LIN {X 52.456,Y -44.205,Z -63.438,A -90.000,B 90.000,C 0.000} C_DIS
LIN {X 52.460,Y -44.237,Z -63.613,A -90.000,B 90.000,C 0.000} C_DIS
LIN {X 52.459,Y -44.265,Z -63.757,A -90.000,B 90.000,C 0.000} C_DIS
LIN {X 52.453,Y -44.312,Z -64.006,A -90.000,B 90.000,C 0.000} C_DIS
LIN {X 52.446,Y -44.340,Z -64.159,A -90.000,B 90.000,C 0.000} C_DIS
LIN {X 52.432,Y -44.368,Z -64.399,A -90.000,B 90.000,C 0.000} C_DIS
LIN {X 52.418,Y -44.378,Z -64.580,A -90.000,B 90.000,C 0.000} C_DIS
LIN {X 52.409,Y -44.383,Z -64.671,A -90.000,B 90.000,C 0.000} C_DIS
LIN {X 52.387,Y -44.391,Z -64.866,A -90.000,B 90.000,C 0.000} C_DIS
LIN {X 52.358,Y -44.401,Z -65.080,A -90.000,B 90.000,C 0.000} C_DIS
LIN {X 52.130,Y -44.481,Z -66.464,A -90.000,B 90.000,C 0.000} C_DIS
LIN {X 52.074,Y -44.507,Z -66.800,A -90.000,B 90.000,C 0.000} C_DIS
LIN {X 52.057,Y -44.512,Z -66.899,A -90.000,B 90.000,C 0.000} C_DIS
LIN {X 52.024,Y -44.517,Z -67.084,A -90.000,B 90.000,C 0.000} C_DIS
LIN {X 51.980,Y -44.511,Z -67.316,A -90.000,B 90.000,C 0.000} C_DIS
LIN {X 51.945,Y -44.501,Z -67.476,A -90.000,B 90.000,C 0.000} C_DIS
LIN {X 51.879,Y -44.478,Z -67.743,A -90.000,B 90.000,C 0.000} C_DIS
LIN {X 51.759,Y -44.433,Z -68.191,A -90.000,B 90.000,C 0.000} C_DIS
LIN {X 51.672,Y -44.408,Z -68.474,A -90.000,B 90.000,C 0.000} C_DIS
LIN {X 51.597,Y -44.391,Z -68.693,A -90.000,B 90.000,C 0.000} C_DIS
LIN {X 51.516,Y -44.382,Z -68.910,A -90.000,B 90.000,C 0.000} C_DIS
LIN {X 51.476,Y -44.378,Z -69.010,A -90.000,B 90.000,C 0.000} C_DIS
LIN {X 51.298,Y -44.364,Z -69.440,A -90.000,B 90.000,C 0.000} C_DIS
LIN {X 51.242,Y -44.352,Z -69.568,A -90.000,B 90.000,C 0.000} C_DIS
LIN {X 51.095,Y -44.326,Z -69.875,A -90.000,B 90.000,C 0.000} C_DIS
LIN {X 50.986,Y -44.297,Z -70.078,A -90.000,B 90.000,C 0.000} C_DIS
LIN {X 50.850,Y -44.249,Z -70.310,A -90.000,B 90.000,C 0.000} C_DIS
LIN {X 50.529,Y -44.147,Z -70.825,A -90.000,B 90.000,C 0.000} C_DIS
LIN {X 50.387,Y -44.107,Z -71.035,A -90.000,B 90.000,C 0.000} C_DIS
LIN {X 50.136,Y -44.044,Z -71.389,A -90.000,B 90.000,C 0.000} C_DIS
LIN {X 49.963,Y -44.011,Z -71.618,A -90.000,B 90.000,C 0.000} C_DIS
LIN {X 49.830,Y -43.988,Z -71.786,A -90.000,B 90.000,C 0.000} C_DIS
LIN {X 49.704,Y -43.961,Z -71.943,A -90.000,B 90.000,C 0.000} C_DIS
LIN {X 49.560,Y -43.918,Z -72.116,A -90.000,B 90.000,C 0.000} C_DIS
LIN {X 49.378,Y -43.866,Z -72.325,A -90.000,B 90.000,C 0.000} C_DIS
LIN {X 49.311,Y -43.846,Z -72.400,A -90.000,B 90.000,C 0.000} C_DIS
LIN {X 48.982,Y -43.733,Z -72.758,A -90.000,B 90.000,C 0.000} C_DIS
LIN {X 48.710,Y -43.636,Z -73.048,A -90.000,B 90.000,C 0.000} C_DIS
LIN {X 48.386,Y -43.521,Z -73.391,A -90.000,B 90.000,C 0.000} C_DIS
LIN {X 48.164,Y -43.447,Z -73.610,A -90.000,B 90.000,C 0.000} C_DIS
LIN {X 47.878,Y -43.351,Z -73.890,A -90.000,B 90.000,C 0.000} C_DIS
LIN {X 47.760,Y -43.308,Z -73.999,A -90.000,B 90.000,C 0.000} C_DIS
LIN {X 47.760,Y -60.000,Z -73.999,A -90.000,B 90.000,C 0.000} C_DIS
LIN {X 54.219,Y -60.000,Z -62.193,A -90.000,B 90.000,C 0.000} C_DIS
LIN {X 54.219,Y -43.308,Z -62.193,A -90.000,B 90.000,C 0.000} C_DIS
LIN {X 54.261,Y -43.356,Z -62.523,A -90.000,B 90.000,C 0.000} C_DIS
LIN {X 54.302,Y -43.419,Z -62.924,A -90.000,B 90.000,C 0.000} C_DIS
LIN {X 54.323,Y -43.471,Z -63.230,A -90.000,B 90.000,C 0.000} C_DIS
LIN {X 54.336,Y -43.540,Z -63.610,A -90.000,B 90.000,C 0.000} C_DIS
LIN {X 54.338,Y -43.581,Z -63.826,A -90.000,B 90.000,C 0.000} C_DIS
LIN {X 54.333,Y -43.640,Z -64.124,A -90.000,B 90.000,C 0.000} C_DIS
LIN {X 54.330,Y -43.665,Z -64.254,A -90.000,B 90.000,C 0.000} C_DIS
LIN {X 54.319,Y -43.710,Z -64.507,A -90.000,B 90.000,C 0.000} C_DIS
LIN {X 54.302,Y -43.748,Z -64.816,A -90.000,B 90.000,C 0.000} C_DIS
LIN {X 54.268,Y -43.772,Z -65.151,A -90.000,B 90.000,C 0.000} C_DIS
LIN {X 54.230,Y -43.786,Z -65.424,A -90.000,B 90.000,C 0.000} C_DIS
LIN {X 53.971,Y -43.885,Z -67.005,A -90.000,B 90.000,C 0.000} C_DIS
LIN {X 53.912,Y -43.907,Z -67.353,A -90.000,B 90.000,C 0.000} C_DIS
LIN {X 53.859,Y -43.908,Z -67.638,A -90.000,B 90.000,C 0.000} C_DIS
LIN {X 53.802,Y -43.893,Z -67.905,A -90.000,B 90.000,C 0.000} C_DIS
LIN {X 53.715,Y -43.863,Z -68.251,A -90.000,B 90.000,C 0.000} C_DIS
LIN {X 53.595,Y -43.826,Z -68.701,A -90.000,B 90.000,C 0.000} C_DIS
LIN {X 53.491,Y -43.802,Z -69.045,A -90.000,B 90.000,C 0.000} C_DIS
LIN {X 53.432,Y -43.792,Z -69.220,A -90.000,B 90.000,C 0.000} C_DIS
LIN {X 53.394,Y -43.791,Z -69.333,A -90.000,B 90.000,C 0.000} C_DIS
LIN {X 53.299,Y -43.790,Z -69.598,A -90.000,B 90.000,C 0.000} C_DIS
LIN {X 53.235,Y -43.791,Z -69.762,A -90.000,B 90.000,C 0.000} C_DIS
LIN {X 53.129,Y -43.778,Z -70.013,A -90.000,B 90.000,C 0.000} C_DIS
LIN {X 53.014,Y -43.746,Z -70.269,A -90.000,B 90.000,C 0.000} C_DIS
LIN {X 52.987,Y -43.738,Z -70.327,A -90.000,B 90.000,C 0.000} C_DIS
LIN {X 52.900,Y -43.714,Z -70.502,A -90.000,B 90.000,C 0.000} C_DIS
LIN {X 52.802,Y -43.680,Z -70.692,A -90.000,B 90.000,C 0.000} C_DIS
LIN {X 52.672,Y -43.639,Z -70.930,A -90.000,B 90.000,C 0.000} C_DIS
LIN {X 52.509,Y -43.592,Z -71.214,A -90.000,B 90.000,C 0.000} C_DIS
LIN {X 52.230,Y -43.521,Z -71.675,A -90.000,B 90.000,C 0.000} C_DIS
LIN {X 52.132,Y -43.504,Z -71.834,A -90.000,B 90.000,C 0.000} C_DIS
LIN {X 52.072,Y -43.495,Z -71.928,A -90.000,B 90.000,C 0.000} C_DIS
LIN {X 51.941,Y -43.468,Z -72.123,A -90.000,B 90.000,C 0.000} C_DIS
LIN {X 51.741,Y -43.423,Z -72.408,A -90.000,B 90.000,C 0.000} C_DIS
LIN {X 51.598,Y -43.382,Z -72.593,A -90.000,B 90.000,C 0.000} C_DIS
LIN {X 51.482,Y -43.343,Z -72.735,A -90.000,B 90.000,C 0.000} C_DIS
LIN {X 51.374,Y -43.308,Z -72.862,A -90.000,B 90.000,C 0.000} C_DIS
LIN {X 51.374,Y -60.000,Z -72.862,A -90.000,B 90.000,C 0.000} C_DIS
LIN {X 38.871,Y -60.000,Z -73.909,A -90.000,B 90.000,C 0.000} C_DIS
LIN {X 38.871,Y -43.308,Z -73.909,A -90.000,B 90.000,C 0.000} C_DIS
LIN {X 38.687,Y -43.323,Z -73.930,A -90.000,B 90.000,C 0.000} C_DIS
LIN {X 38.483,Y -43.337,Z -73.949,A -90.000,B 90.000,C 0.000} C_DIS
LIN {X 38.230,Y -43.361,Z -73.961,A -90.000,B 90.000,C 0.000} C_DIS
LIN {X 38.066,Y -43.380,Z -73.963,A -90.000,B 90.000,C 0.000} C_DIS
LIN {X 37.937,Y -43.397,Z -73.961,A -90.000,B 90.000,C 0.000} C_DIS
LIN {X 37.611,Y -43.421,Z -73.939,A -90.000,B 90.000,C 0.000} C_DIS
LIN {X 37.303,Y -43.447,Z -73.906,A -90.000,B 90.000,C 0.000} C_DIS
LIN {X 36.954,Y -43.483,Z -73.874,A -90.000,B 90.000,C 0.000} C_DIS
LIN {X 36.730,Y -43.505,Z -73.852,A -90.000,B 90.000,C 0.000} C_DIS
LIN {X 36.470,Y -43.514,Z -73.811,A -90.000,B 90.000,C 0.000} C_DIS
LIN {X 36.378,Y -43.519,Z -73.793,A -90.000,B 90.000,C 0.000} C_DIS
LIN {X 36.077,Y -43.530,Z -73.720,A -90.000,B 90.000,C 0.000} C_DIS
LIN {X 35.883,Y -43.539,Z -73.671,A -90.000,B 90.000,C 0.000} C_DIS
LIN {X 35.758,Y -43.548,Z -73.635,A -90.000,B 90.000,C 0.000} C_DIS
LIN {X 35.646,Y -43.559,Z -73.599,A -90.000,B 90.000,C 0.000} C_DIS
LIN {X 35.484,Y -43.570,Z -73.540,A -90.000,B 90.000,C 0.000} C_DIS
LIN {X 35.327,Y -43.582,Z -73.478,A -90.000,B 90.000,C 0.000} C_DIS
LIN {X 35.176,Y -43.589,Z -73.417,A -90.000,B 90.000,C 0.000} C_DIS
LIN {X 34.989,Y -43.592,Z -73.329,A -90.000,B 90.000,C 0.000} C_DIS
LIN {X 34.877,Y -43.596,Z -73.270,A -90.000,B 90.000,C 0.000} C_DIS
LIN {X 34.689,Y -43.603,Z -73.162,A -90.000,B 90.000,C 0.000} C_DIS
LIN {X 34.340,Y -43.621,Z -72.948,A -90.000,B 90.000,C 0.000} C_DIS
LIN {X 34.071,Y -43.622,Z -72.775,A -90.000,B 90.000,C 0.000} C_DIS
LIN {X 33.848,Y -43.608,Z -72.620,A -90.000,B 90.000,C 0.000} C_DIS
LIN {X 33.739,Y -43.595,Z -72.541,A -90.000,B 90.000,C 0.000} C_DIS
LIN {X 33.578,Y -43.580,Z -72.414,A -90.000,B 90.000,C 0.000} C_DIS
LIN {X 33.361,Y -43.557,Z -72.215,A -90.000,B 90.000,C 0.000} C_DIS
LIN {X 33.169,Y -43.538,Z -72.034,A -90.000,B 90.000,C 0.000} C_DIS
LIN {X 33.088,Y -43.529,Z -71.950,A -90.000,B 90.000,C 0.000} C_DIS
LIN {X 32.980,Y -43.517,Z -71.834,A -90.000,B 90.000,C 0.000} C_DIS
LIN {X 32.939,Y -43.514,Z -71.787,A -90.000,B 90.000,C 0.000} C_DIS
LIN {X 32.866,Y -43.500,Z -71.695,A -90.000,B 90.000,C 0.000} C_DIS
LIN {X 32.747,Y -43.481,Z -71.535,A -90.000,B 90.000,C 0.000} C_DIS
LIN {X 32.592,Y -43.443,Z -71.305,A -90.000,B 90.000,C 0.000} C_DIS
LIN {X 32.502,Y -43.419,Z -71.160,A -90.000,B 90.000,C 0.000} C_DIS
LIN {X 32.424,Y -43.400,Z -71.023,A -90.000,B 90.000,C 0.000} C_DIS
LIN {X 32.315,Y -43.356,Z -70.787,A -90.000,B 90.000,C 0.000} C_DIS
LIN {X 32.203,Y -43.308,Z -70.519,A -90.000,B 90.000,C 0.000} C_DIS
LIN {X 32.203,Y -60.000,Z -70.519,A -90.000,B 90.000,C 0.000} C_DIS
LIN {X 37.582,Y -60.000,Z -56.436,A -90.000,B 90.000,C 0.000} C_DIS
LIN {X 37.582,Y -43.308,Z -56.436,A -90.000,B 90.000,C 0.000} C_DIS
LIN {X 37.821,Y -43.324,Z -56.331,A -90.000,B 90.000,C 0.000} C_DIS
LIN {X 37.931,Y -43.333,Z -56.286,A -90.000,B 90.000,C 0.000} C_DIS
LIN {X 38.127,Y -43.352,Z -56.209,A -90.000,B 90.000,C 0.000} C_DIS
LIN {X 38.445,Y -43.384,Z -56.093,A -90.000,B 90.000,C 0.000} C_DIS
LIN {X 38.740,Y -43.393,Z -56.001,A -90.000,B 90.000,C 0.000} C_DIS
LIN {X 38.778,Y -43.395,Z -55.990,A -90.000,B 90.000,C 0.000} C_DIS
LIN {X 39.258,Y -43.388,Z -55.877,A -90.000,B 90.000,C 0.000} C_DIS
LIN {X 39.652,Y -43.384,Z -55.789,A -90.000,B 90.000,C 0.000} C_DIS
LIN {X 39.801,Y -43.386,Z -55.761,A -90.000,B 90.000,C 0.000} C_DIS
LIN {X 39.916,Y -43.388,Z -55.741,A -90.000,B 90.000,C 0.000} C_DIS
LIN {X 40.073,Y -43.394,Z -55.720,A -90.000,B 90.000,C 0.000} C_DIS
LIN {X 40.424,Y -43.393,Z -55.695,A -90.000,B 90.000,C 0.000} C_DIS
LIN {X 40.588,Y -43.382,Z -55.692,A -90.000,B 90.000,C 0.000} C_DIS
LIN {X 40.769,Y -43.375,Z -55.695,A -90.000,B 90.000,C 0.000} C_DIS
LIN {X 40.998,Y -43.363,Z -55.713,A -90.000,B 90.000,C 0.000} C_DIS
LIN {X 41.338,Y -43.351,Z -55.748,A -90.000,B 90.000,C 0.000} C_DIS
LIN {X 41.531,Y -43.350,Z -55.776,A -90.000,B 90.000,C 0.000} C_DIS
LIN {X 41.746,Y -43.351,Z -55.811,A -90.000,B 90.000,C 0.000} C_DIS
LIN {X 41.864,Y -43.353,Z -55.835,A -90.000,B 90.000,C 0.000} C_DIS
LIN {X 42.226,Y -43.361,Z -55.917,A -90.000,B 90.000,C 0.000} C_DIS
LIN {X 42.582,Y -43.346,Z -56.012,A -90.000,B 90.000,C 0.000} C_DIS
LIN {X 42.854,Y -43.316,Z -56.101,A -90.000,B 90.000,C 0.000} C_DIS
LIN {X 42.925,Y -43.308,Z -56.126,A -90.000,B 90.000,C 0.000} C_DIS
LIN {X 43.177,Y -43.308,Z -56.261,A -90.000,B 90.000,C 0.000} C_DIS
LIN {X 43.997,Y -43.308,Z -56.741,A -90.000,B 90.000,C 0.000} C_DIS
LIN {X 44.082,Y -43.308,Z -56.794,A -90.000,B 90.000,C 0.000} C_DIS
LIN {X 44.337,Y -43.308,Z -56.962,A -90.000,B 90.000,C 0.000} C_DIS
LIN {X 44.400,Y -43.308,Z -57.009,A -90.000,B 90.000,C 0.000} C_DIS
LIN {X 44.745,Y -43.308,Z -57.308,A -90.000,B 90.000,C 0.000} C_DIS
LIN {X 45.353,Y -43.308,Z -57.963,A -90.000,B 90.000,C 0.000} C_DIS
LIN {X 45.605,Y -43.308,Z -58.247,A -90.000,B 90.000,C 0.000} C_DIS
LIN {X 45.739,Y -43.308,Z -58.416,A -90.000,B 90.000,C 0.000} C_DIS
LIN {X 46.082,Y -43.308,Z -58.777,A -90.000,B 90.000,C 0.000} C_DIS
LIN {X 46.305,Y -43.308,Z -59.042,A -90.000,B 90.000,C 0.000} C_DIS
LIN {X 46.345,Y -43.308,Z -59.069,A -90.000,B 90.000,C 0.000} C_DIS
LIN {X 46.450,Y -43.308,Z -59.152,A -90.000,B 90.000,C 0.000} C_DIS
LIN {X 46.761,Y -43.308,Z -59.167,A -90.000,B 90.000,C 0.000} C_DIS
LIN {X 47.921,Y -43.308,Z -58.993,A -90.000,B 90.000,C 0.000} C_DIS
LIN {X 48.239,Y -43.308,Z -58.971,A -90.000,B 90.000,C 0.000} C_DIS
LIN {X 49.722,Y -43.308,Z -58.969,A -90.000,B 90.000,C 0.000} C_DIS
LIN {X 50.041,Y -43.308,Z -58.996,A -90.000,B 90.000,C 0.000} C_DIS
LIN {X 50.351,Y -43.308,Z -59.073,A -90.000,B 90.000,C 0.000} C_DIS
LIN {X 50.521,Y -43.308,Z -59.144,A -90.000,B 90.000,C 0.000} C_DIS
LIN {X 51.662,Y -43.308,Z -59.634,A -90.000,B 90.000,C 0.000} C_DIS
LIN {X 52.223,Y -43.308,Z -59.869,A -90.000,B 90.000,C 0.000} C_DIS
LIN {X 52.495,Y -43.308,Z -60.037,A -90.000,B 90.000,C 0.000} C_DIS
LIN {X 52.737,Y -43.308,Z -60.246,A -90.000,B 90.000,C 0.000} C_DIS
LIN {X 52.843,Y -43.308,Z -60.348,A -90.000,B 90.000,C 0.000} C_DIS
LIN {X 53.100,Y -43.308,Z -60.607,A -90.000,B 90.000,C 0.000} C_DIS
LIN {X 53.314,Y -43.308,Z -60.850,A -90.000,B 90.000,C 0.000} C_DIS
LIN {X 53.845,Y -43.308,Z -61.517,A -90.000,B 90.000,C 0.000} C_DIS
LIN {X 54.011,Y -43.308,Z -61.790,A -90.000,B 90.000,C 0.000} C_DIS
LIN {X 54.321,Y -43.308,Z -62.391,A -90.000,B 90.000,C 0.000} C_DIS
LIN {X 54.587,Y -43.308,Z -62.899,A -90.000,B 90.000,C 0.000} C_DIS
LIN {X 54.709,Y -43.308,Z -63.195,A -90.000,B 90.000,C 0.000} C_DIS
LIN {X 55.026,Y -43.308,Z -64.144,A -90.000,B 90.000,C 0.000} C_DIS
LIN {X 55.237,Y -43.308,Z -64.763,A -90.000,B 90.000,C 0.000} C_DIS
LIN {X 55.311,Y -43.308,Z -65.074,A -90.000,B 90.000,C 0.000} C_DIS
LIN {X 55.336,Y -43.308,Z -65.392,A -90.000,B 90.000,C 0.000} C_DIS
LIN {X 55.335,Y -43.308,Z -65.444,A -90.000,B 90.000,C 0.000} C_DIS
LIN {X 55.311,Y -43.308,Z -66.357,A -90.000,B 90.000,C 0.000} C_DIS
LIN {X 55.366,Y -43.308,Z -67.491,A -90.000,B 90.000,C 0.000} C_DIS
LIN {X 55.366,Y -43.308,Z -67.611,A -90.000,B 90.000,C 0.000} C_DIS
LIN {X 55.361,Y -43.308,Z -67.740,A -90.000,B 90.000,C 0.000} C_DIS
LIN {X 55.313,Y -43.308,Z -68.018,A -90.000,B 90.000,C 0.000} C_DIS
LIN {X 55.218,Y -43.308,Z -68.283,A -90.000,B 90.000,C 0.000} C_DIS
LIN {X 54.561,Y -43.308,Z -70.046,A -90.000,B 90.000,C 0.000} C_DIS
LIN {X 54.420,Y -43.308,Z -70.290,A -90.000,B 90.000,C 0.000} C_DIS
LIN {X 54.238,Y -43.308,Z -70.507,A -90.000,B 90.000,C 0.000} C_DIS
LIN {X 54.016,Y -43.308,Z -70.742,A -90.000,B 90.000,C 0.000} C_DIS
LIN {X 53.865,Y -43.308,Z -70.875,A -90.000,B 90.000,C 0.000} C_DIS
LIN {X 52.680,Y -43.308,Z -72.037,A -90.000,B 90.000,C 0.000} C_DIS
LIN {X 52.463,Y -43.308,Z -72.217,A -90.000,B 90.000,C 0.000} C_DIS
LIN {X 52.116,Y -43.308,Z -72.476,A -90.000,B 90.000,C 0.000} C_DIS
LIN {X 51.840,Y -43.308,Z -72.637,A -90.000,B 90.000,C 0.000} C_DIS
LIN {X 51.007,Y -43.308,Z -73.039,A -90.000,B 90.000,C 0.000} C_DIS
LIN {X 50.709,Y -43.308,Z -73.155,A -90.000,B 90.000,C 0.000} C_DIS
LIN {X 48.918,Y -43.308,Z -73.715,A -90.000,B 90.000,C 0.000} C_DIS
LIN {X 48.353,Y -43.308,Z -73.902,A -90.000,B 90.000,C 0.000} C_DIS
LIN {X 48.041,Y -43.308,Z -73.971,A -90.000,B 90.000,C 0.000} C_DIS
LIN {X 47.916,Y -43.308,Z -73.990,A -90.000,B 90.000,C 0.000} C_DIS
LIN {X 47.687,Y -43.308,Z -74.003,A -90.000,B 90.000,C 0.000} C_DIS
LIN {X 47.607,Y -43.308,Z -74.002,A -90.000,B 90.000,C 0.000} C_DIS
LIN {X 46.022,Y -43.308,Z -73.914,A -90.000,B 90.000,C 0.000} C_DIS
LIN {X 45.594,Y -43.308,Z -73.873,A -90.000,B 90.000,C 0.000} C_DIS
LIN {X 45.317,Y -43.308,Z -73.819,A -90.000,B 90.000,C 0.000} C_DIS
LIN {X 44.160,Y -43.308,Z -73.448,A -90.000,B 90.000,C 0.000} C_DIS
LIN {X 43.984,Y -43.308,Z -73.397,A -90.000,B 90.000,C 0.000} C_DIS
LIN {X 43.751,Y -43.308,Z -73.306,A -90.000,B 90.000,C 0.000} C_DIS
LIN {X 43.025,Y -43.308,Z -72.995,A -90.000,B 90.000,C 0.000} C_DIS
LIN {X 42.728,Y -43.308,Z -72.850,A -90.000,B 90.000,C 0.000} C_DIS
LIN {X 42.198,Y -43.308,Z -72.717,A -90.000,B 90.000,C 0.000} C_DIS
LIN {X 41.959,Y -43.308,Z -72.770,A -90.000,B 90.000,C 0.000} C_DIS
LIN {X 41.917,Y -43.308,Z -72.792,A -90.000,B 90.000,C 0.000} C_DIS
LIN {X 40.967,Y -43.308,Z -73.176,A -90.000,B 90.000,C 0.000} C_DIS
LIN {X 40.944,Y -43.308,Z -73.188,A -90.000,B 90.000,C 0.000} C_DIS
LIN {X 40.456,Y -43.308,Z -73.390,A -90.000,B 90.000,C 0.000} C_DIS
LIN {X 40.263,Y -43.308,Z -73.467,A -90.000,B 90.000,C 0.000} C_DIS
LIN {X 39.930,Y -43.308,Z -73.593,A -90.000,B 90.000,C 0.000} C_DIS
LIN {X 39.677,Y -43.308,Z -73.675,A -90.000,B 90.000,C 0.000} C_DIS
LIN {X 39.567,Y -43.308,Z -73.702,A -90.000,B 90.000,C 0.000} C_DIS
LIN {X 39.007,Y -43.308,Z -73.876,A -90.000,B 90.000,C 0.000} C_DIS
LIN {X 38.761,Y -43.308,Z -73.937,A -90.000,B 90.000,C 0.000} C_DIS
LIN {X 38.686,Y -43.308,Z -73.953,A -90.000,B 90.000,C 0.000} C_DIS
LIN {X 37.844,Y -43.308,Z -74.113,A -90.000,B 90.000,C 0.000} C_DIS
LIN {X 37.519,Y -43.308,Z -74.129,A -90.000,B 90.000,C 0.000} C_DIS
LIN {X 37.008,Y -43.308,Z -74.148,A -90.000,B 90.000,C 0.000} C_DIS
LIN {X 36.887,Y -43.308,Z -74.158,A -90.000,B 90.000,C 0.000} C_DIS
LIN {X 36.536,Y -43.308,Z -74.176,A -90.000,B 90.000,C 0.000} C_DIS
LIN {X 36.186,Y -43.308,Z -74.145,A -90.000,B 90.000,C 0.000} C_DIS
LIN {X 35.524,Y -43.308,Z -74.028,A -90.000,B 90.000,C 0.000} C_DIS
LIN {X 35.410,Y -43.308,Z -74.011,A -90.000,B 90.000,C 0.000} C_DIS
LIN {X 35.068,Y -43.308,Z -73.930,A -90.000,B 90.000,C 0.000} C_DIS
LIN {X 34.983,Y -43.308,Z -73.903,A -90.000,B 90.000,C 0.000} C_DIS
LIN {X 34.847,Y -43.308,Z -73.849,A -90.000,B 90.000,C 0.000} C_DIS
LIN {X 34.676,Y -43.308,Z -73.775,A -90.000,B 90.000,C 0.000} C_DIS
LIN {X 34.113,Y -43.308,Z -73.493,A -90.000,B 90.000,C 0.000} C_DIS
LIN {X 33.942,Y -43.308,Z -73.395,A -90.000,B 90.000,C 0.000} C_DIS
LIN {X 33.823,Y -43.308,Z -73.320,A -90.000,B 90.000,C 0.000} C_DIS
LIN {X 33.668,Y -43.308,Z -73.199,A -90.000,B 90.000,C 0.000} C_DIS
LIN {X 33.575,Y -43.308,Z -73.121,A -90.000,B 90.000,C 0.000} C_DIS
LIN {X 33.331,Y -43.308,Z -72.868,A -90.000,B 90.000,C 0.000} C_DIS
LIN {X 32.968,Y -43.308,Z -72.431,A -90.000,B 90.000,C 0.000} C_DIS
LIN {X 32.762,Y -43.308,Z -72.146,A -90.000,B 90.000,C 0.000} C_DIS
LIN {X 32.598,Y -43.308,Z -71.835,A -90.000,B 90.000,C 0.000} C_DIS
LIN {X 32.475,Y -43.308,Z -71.537,A -90.000,B 90.000,C 0.000} C_DIS
LIN {X 32.344,Y -43.308,Z -71.181,A -90.000,B 90.000,C 0.000} C_DIS
LIN {X 32.265,Y -43.308,Z -70.832,A -90.000,B 90.000,C 0.000} C_DIS
LIN {X 32.198,Y -43.308,Z -70.496,A -90.000,B 90.000,C 0.000} C_DIS
LIN {X 32.059,Y -43.308,Z -69.876,A -90.000,B 90.000,C 0.000} C_DIS
LIN {X 32.000,Y -43.308,Z -69.477,A -90.000,B 90.000,C 0.000} C_DIS
LIN {X 31.983,Y -43.308,Z -69.251,A -90.000,B 90.000,C 0.000} C_DIS
LIN {X 31.977,Y -43.308,Z -68.971,A -90.000,B 90.000,C 0.000} C_DIS
LIN {X 31.978,Y -43.308,Z -68.841,A -90.000,B 90.000,C 0.000} C_DIS
LIN {X 31.999,Y -43.308,Z -68.128,A -90.000,B 90.000,C 0.000} C_DIS
LIN {X 32.033,Y -43.308,Z -67.741,A -90.000,B 90.000,C 0.000} C_DIS
LIN {X 32.067,Y -43.308,Z -67.060,A -90.000,B 90.000,C 0.000} C_DIS
LIN {X 32.121,Y -43.308,Z -66.651,A -90.000,B 90.000,C 0.000} C_DIS
LIN {X 32.359,Y -43.308,Z -65.353,A -90.000,B 90.000,C 0.000} C_DIS
LIN {X 32.466,Y -43.308,Z -64.935,A -90.000,B 90.000,C 0.000} C_DIS
LIN {X 32.831,Y -43.308,Z -63.566,A -90.000,B 90.000,C 0.000} C_DIS
LIN {X 32.944,Y -43.308,Z -63.220,A -90.000,B 90.000,C 0.000} C_DIS
LIN {X 33.474,Y -43.308,Z -61.799,A -90.000,B 90.000,C 0.000} C_DIS
LIN {X 34.220,Y -43.308,Z -60.166,A -90.000,B 90.000,C 0.000} C_DIS
LIN {X 34.404,Y -43.308,Z -59.808,A -90.000,B 90.000,C 0.000} C_DIS
LIN {X 34.871,Y -43.308,Z -59.121,A -90.000,B 90.000,C 0.000} C_DIS
LIN {X 35.174,Y -43.308,Z -58.706,A -90.000,B 90.000,C 0.000} C_DIS
LIN {X 35.553,Y -43.308,Z -58.179,A -90.000,B 90.000,C 0.000} C_DIS
LIN {X 35.797,Y -43.308,Z -57.889,A -90.000,B 90.000,C 0.000} C_DIS
LIN {X 36.217,Y -43.308,Z -57.462,A -90.000,B 90.000,C 0.000} C_DIS
LIN {X 36.362,Y -43.308,Z -57.331,A -90.000,B 90.000,C 0.000} C_DIS
LIN {X 36.781,Y -43.308,Z -56.955,A -90.000,B 90.000,C 0.000} C_DIS
LIN {X 36.859,Y -43.308,Z -56.885,A -90.000,B 90.000,C 0.000} C_DIS
LIN {X 37.171,Y -43.308,Z -56.669,A -90.000,B 90.000,C 0.000} C_DIS
LIN {X 37.236,Y -43.308,Z -56.630,A -90.000,B 90.000,C 0.000} C_DIS
LIN {X 37.735,Y -43.308,Z -56.351,A -90.000,B 90.000,C 0.000} C_DIS
LIN {X 38.116,Y -43.308,Z -56.142,A -90.000,B 90.000,C 0.000} C_DIS
LIN {X 38.425,Y -43.308,Z -55.976,A -90.000,B 90.000,C 0.000} C_DIS
LIN {X 38.756,Y -43.308,Z -55.856,A -90.000,B 90.000,C 0.000} C_DIS
LIN {X 39.336,Y -43.308,Z -55.733,A -90.000,B 90.000,C 0.000} C_DIS
LIN {X 40.049,Y -43.308,Z -55.588,A -90.000,B 90.000,C 0.000} C_DIS
LIN {X 40.400,Y -43.308,Z -55.565,A -90.000,B 90.000,C 0.000} C_DIS
LIN {X 40.751,Y -43.308,Z -55.592,A -90.000,B 90.000,C 0.000} C_DIS
LIN {X 41.785,Y -43.308,Z -55.753,A -90.000,B 90.000,C 0.000} C_DIS
LIN {X 42.212,Y -43.308,Z -55.836,A -90.000,B 90.000,C 0.000} C_DIS
LIN {X 42.572,Y -43.308,Z -55.955,A -90.000,B 90.000,C 0.000} C_DIS
LIN {X 42.913,Y -43.308,Z -56.120,A -90.000,B 90.000,C 0.000} C_DIS
LIN {X 42.925,Y -43.308,Z -56.126,A -90.000,B 90.000,C 0.000} C_DIS
LIN {X 42.925,Y -60.000,Z -56.126,A -90.000,B 90.000,C 0.000} C_DIS
LIN {X 52.003,Y -60.000,Z -168.388,A -90.000,B 90.000,C 0.000} C_DIS
LIN {X 52.003,Y -47.267,Z -168.388,A -90.000,B 90.000,C 0.000} C_DIS
LIN {X 52.090,Y -47.269,Z -168.387,A -90.000,B 90.000,C 0.000} C_DIS
LIN {X 52.222,Y -47.274,Z -168.394,A -90.000,B 90.000,C 0.000} C_DIS
LIN {X 52.299,Y -47.277,Z -168.401,A -90.000,B 90.000,C 0.000} C_DIS
LIN {X 52.434,Y -47.282,Z -168.422,A -90.000,B 90.000,C 0.000} C_DIS
LIN {X 52.499,Y -47.284,Z -168.435,A -90.000,B 90.000,C 0.000} C_DIS
LIN {X 52.623,Y -47.286,Z -168.467,A -90.000,B 90.000,C 0.000} C_DIS
LIN {X 52.723,Y -47.286,Z -168.499,A -90.000,B 90.000,C 0.000} C_DIS
LIN {X 52.840,Y -47.283,Z -168.544,A -90.000,B 90.000,C 0.000} C_DIS
LIN {X 52.993,Y -47.276,Z -168.617,A -90.000,B 90.000,C 0.000} C_DIS
LIN {X 53.188,Y -47.266,Z -168.734,A -90.000,B 90.000,C 0.000} C_DIS
LIN {X 53.273,Y -47.262,Z -168.795,A -90.000,B 90.000,C 0.000} C_DIS
LIN {X 53.360,Y -47.258,Z -168.865,A -90.000,B 90.000,C 0.000} C_DIS
LIN {X 53.483,Y -47.252,Z -168.980,A -90.000,B 90.000,C 0.000} C_DIS
LIN {X 53.605,Y -47.246,Z -169.115,A -90.000,B 90.000,C 0.000} C_DIS
LIN {X 53.692,Y -47.242,Z -169.228,A -90.000,B 90.000,C 0.000} C_DIS
LIN {X 53.735,Y -47.240,Z -169.292,A -90.000,B 90.000,C 0.000} C_DIS
LIN {X 53.821,Y -47.235,Z -169.436,A -90.000,B 90.000,C 0.000} C_DIS
LIN {X 53.911,Y -47.229,Z -169.627,A -90.000,B 90.000,C 0.000} C_DIS
LIN {X 54.002,Y -47.222,Z -169.875,A -90.000,B 90.000,C 0.000} C_DIS
LIN {X 54.042,Y -47.220,Z -169.998,A -90.000,B 90.000,C 0.000} C_DIS
LIN {X 54.066,Y -47.218,Z -170.083,A -90.000,B 90.000,C 0.000} C_DIS
LIN {X 54.098,Y -47.215,Z -170.211,A -90.000,B 90.000,C 0.000} C_DIS
LIN {X 54.142,Y -47.209,Z -170.704,A -90.000,B 90.000,C 0.000} C_DIS
LIN {X 54.133,Y -47.208,Z -170.835,A -90.000,B 90.000,C 0.000} C_DIS
LIN {X 54.055,Y -47.205,Z -171.617,A -90.000,B 90.000,C 0.000} C_DIS
LIN {X 53.987,Y -47.204,Z -172.285,A -90.000,B 90.000,C 0.000} C_DIS
LIN {X 53.992,Y -47.203,Z -172.639,A -90.000,B 90.000,C 0.000} C_DIS
LIN {X 53.982,Y -47.205,Z -174.437,A -90.000,B 90.000,C 0.000} C_DIS
LIN {X 53.978,Y -47.200,Z -174.947,A -90.000,B 90.000,C 0.000} C_DIS
LIN {X 54.085,Y -47.186,Z -175.467,A -90.000,B 90.000,C 0.000} C_DIS
LIN {X 54.450,Y -47.135,Z -177.245,A -90.000,B 90.000,C 0.000} C_DIS
LIN {X 54.473,Y -47.132,Z -177.381,A -90.000,B 90.000,C 0.000} C_DIS
LIN {X 54.481,Y -47.130,Z -177.446,A -90.000,B 90.000,C 0.000} C_DIS
LIN {X 54.517,Y -47.126,Z -177.536,A -90.000,B 90.000,C 0.000} C_DIS
LIN {X 54.562,Y -47.120,Z -177.676,A -90.000,B 90.000,C 0.000} C_DIS
LIN {X 54.587,Y -47.117,Z -177.761,A -90.000,B 90.000,C 0.000} C_DIS
LIN {X 54.655,Y -47.107,Z -178.136,A -90.000,B 90.000,C 0.000} C_DIS
LIN {X 54.670,Y -47.104,Z -178.310,A -90.000,B 90.000,C 0.000} C_DIS
LIN {X 54.753,Y -47.105,Z -179.245,A -90.000,B 90.000,C 0.000} C_DIS
LIN {X 54.760,Y -47.106,Z -179.363,A -90.000,B 90.000,C 0.000} C_DIS
LIN {X 54.779,Y -47.111,Z -180.008,A -90.000,B 90.000,C 0.000} C_DIS
LIN {X 54.789,Y -47.112,Z -180.335,A -90.000,B 90.000,C 0.000} C_DIS
LIN {X 54.861,Y -47.106,Z -180.697,A -90.000,B 90.000,C 0.000} C_DIS
LIN {X 54.880,Y -47.105,Z -180.811,A -90.000,B 90.000,C 0.000} C_DIS
LIN {X 54.898,Y -47.103,Z -180.943,A -90.000,B 90.000,C 0.000} C_DIS
LIN {X 55.064,Y -47.114,Z -182.341,A -90.000,B 90.000,C 0.000} C_DIS
LIN {X 55.111,Y -47.110,Z -182.742,A -90.000,B 90.000,C 0.000} C_DIS
LIN {X 55.344,Y -47.078,Z -183.664,A -90.000,B 90.000,C 0.000} C_DIS
LIN {X 55.573,Y -47.057,Z -184.570,A -90.000,B 90.000,C 0.000} C_DIS
LIN {X 55.680,Y -47.045,Z -184.995,A -90.000,B 90.000,C 0.000} C_DIS
LIN {X 55.762,Y -47.035,Z -185.329,A -90.000,B 90.000,C 0.000} C_DIS
LIN {X 55.797,Y -47.031,Z -185.515,A -90.000,B 90.000,C 0.000} C_DIS
LIN {X 55.822,Y -47.029,Z -185.693,A -90.000,B 90.000,C 0.000} C_DIS
LIN {X 55.840,Y -47.027,Z -185.915,A -90.000,B 90.000,C 0.000} C_DIS
LIN {X 55.850,Y -47.028,Z -186.301,A -90.000,B 90.000,C 0.000} C_DIS
LIN {X 55.909,Y -47.043,Z -188.434,A -90.000,B 90.000,C 0.000} C_DIS
LIN {X 55.936,Y -47.044,Z -189.714,A -90.000,B 90.000,C 0.000} C_DIS
LIN {X 55.936,Y -47.044,Z -189.794,A -90.000,B 90.000,C 0.000} C_DIS
LIN {X 55.923,Y -47.047,Z -190.433,A -90.000,B 90.000,C 0.000} C_DIS
LIN {X 55.898,Y -47.032,Z -191.546,A -90.000,B 90.000,C 0.000} C_DIS
LIN {X 55.873,Y -47.029,Z -191.995,A -90.000,B 90.000,C 0.000} C_DIS
LIN {X 55.731,Y -46.980,Z -194.310,A -90.000,B 90.000,C 0.000} C_DIS
LIN {X 55.662,Y -46.967,Z -195.095,A -90.000,B 90.000,C 0.000} C_DIS
LIN {X 55.642,Y -46.966,Z -195.251,A -90.000,B 90.000,C 0.000} C_DIS
LIN {X 55.576,Y -46.962,Z -195.638,A -90.000,B 90.000,C 0.000} C_DIS
LIN {X 55.371,Y -46.935,Z -197.090,A -90.000,B 90.000,C 0.000} C_DIS
LIN {X 55.334,Y -46.933,Z -197.286,A -90.000,B 90.000,C 0.000} C_DIS
LIN {X 55.099,Y -46.933,Z -198.249,A -90.000,B 90.000,C 0.000} C_DIS
LIN {X 54.880,Y -46.933,Z -199.148,A -90.000,B 90.000,C 0.000} C_DIS
LIN {X 54.849,Y -46.932,Z -199.269,A -90.000,B 90.000,C 0.000} C_DIS
LIN {X 54.182,Y -46.935,Z -201.573,A -90.000,B 90.000,C 0.000} C_DIS
LIN {X 53.558,Y -46.935,Z -203.721,A -90.000,B 90.000,C 0.000} C_DIS
LIN {X 53.350,Y -46.935,Z -204.388,A -90.000,B 90.000,C 0.000} C_DIS
LIN {X 52.108,Y -46.938,Z -208.275,A -90.000,B 90.000,C 0.000} C_DIS
LIN {X 51.309,Y -46.938,Z -210.719,A -90.000,B 90.000,C 0.000} C_DIS
LIN {X 50.451,Y -46.943,Z -213.262,A -90.000,B 90.000,C 0.000} C_DIS
LIN {X 49.740,Y -46.948,Z -215.306,A -90.000,B 90.000,C 0.000} C_DIS
LIN {X 48.678,Y -46.909,Z -218.520,A -90.000,B 90.000,C 0.000} C_DIS
LIN {X 48.628,Y -46.907,Z -218.653,A -90.000,B 90.000,C 0.000} C_DIS
LIN {X 48.118,Y -46.903,Z -219.874,A -90.000,B 90.000,C 0.000} C_DIS
LIN {X 47.332,Y -46.884,Z -221.874,A -90.000,B 90.000,C 0.000} C_DIS
LIN {X 46.592,Y -46.868,Z -223.757,A -90.000,B 90.000,C 0.000} C_DIS
LIN {X 46.503,Y -46.862,Z -223.973,A -90.000,B 90.000,C 0.000} C_DIS
LIN {X 46.426,Y -46.861,Z -224.129,A -90.000,B 90.000,C 0.000} C_DIS
LIN {X 46.088,Y -46.864,Z -224.740,A -90.000,B 90.000,C 0.000} C_DIS
LIN {X 44.574,Y -46.859,Z -227.627,A -90.000,B 90.000,C 0.000} C_DIS
LIN {X 43.772,Y -46.861,Z -229.159,A -90.000,B 90.000,C 0.000} C_DIS
LIN {X 43.723,Y -46.858,Z -229.251,A -90.000,B 90.000,C 0.000} C_DIS
LIN {X 43.624,Y -46.854,Z -229.419,A -90.000,B 90.000,C 0.000} C_DIS
LIN {X 43.526,Y -46.853,Z -229.569,A -90.000,B 90.000,C 0.000} C_DIS
LIN {X 43.424,Y -46.853,Z -229.711,A -90.000,B 90.000,C 0.000} C_DIS
LIN {X 42.952,Y -46.866,Z -230.315,A -90.000,B 90.000,C 0.000} C_DIS
LIN {X 40.607,Y -46.909,Z -233.434,A -90.000,B 90.000,C 0.000} C_DIS
LIN {X 40.134,Y -46.921,Z -234.065,A -90.000,B 90.000,C 0.000} C_DIS
LIN {X 40.008,Y -46.919,Z -234.230,A -90.000,B 90.000,C 0.000} C_DIS
LIN {X 39.772,Y -46.908,Z -234.540,A -90.000,B 90.000,C 0.000} C_DIS
LIN {X 39.720,Y -46.906,Z -234.604,A -90.000,B 90.000,C 0.000} C_DIS
LIN {X 39.528,Y -46.906,Z -234.806,A -90.000,B 90.000,C 0.000} C_DIS
LIN {X 39.247,Y -46.914,Z -235.063,A -90.000,B 90.000,C 0.000} C_DIS
LIN {X 38.633,Y -46.940,Z -235.585,A -90.000,B 90.000,C 0.000} C_DIS
LIN {X 37.370,Y -46.946,Z -236.649,A -90.000,B 90.000,C 0.000} C_DIS
LIN {X 36.098,Y -46.950,Z -237.720,A -90.000,B 90.000,C 0.000} C_DIS
LIN {X 35.251,Y -46.950,Z -238.452,A -90.000,B 90.000,C 0.000} C_DIS
LIN {X 34.978,Y -46.947,Z -238.687,A -90.000,B 90.000,C 0.000} C_DIS
LIN {X 34.342,Y -46.925,Z -239.232,A -90.000,B 90.000,C 0.000} C_DIS
LIN {X 34.228,Y -46.922,Z -239.322,A -90.000,B 90.000,C 0.000} C_DIS
LIN {X 33.933,Y -46.917,Z -239.539,A -90.000,B 90.000,C 0.000} C_DIS
LIN {X 33.825,Y -46.917,Z -239.614,A -90.000,B 90.000,C 0.000} C_DIS
LIN {X 32.960,Y -46.917,Z -240.168,A -90.000,B 90.000,C 0.000} C_DIS
LIN {X 31.948,Y -46.921,Z -240.788,A -90.000,B 90.000,C 0.000} C_DIS
LIN {X 31.798,Y -46.924,Z -240.871,A -90.000,B 90.000,C 0.000} C_DIS
LIN {X 31.609,Y -46.929,Z -240.961,A -90.000,B 90.000,C 0.000} C_DIS
LIN {X 31.405,Y -46.936,Z -241.047,A -90.000,B 90.000,C 0.000} C_DIS
LIN {X 29.828,Y -47.012,Z -241.606,A -90.000,B 90.000,C 0.000} C_DIS
LIN {X 28.974,Y -47.049,Z -241.907,A -90.000,B 90.000,C 0.000} C_DIS
LIN {X 28.817,Y -47.052,Z -241.962,A -90.000,B 90.000,C 0.000} C_DIS
LIN {X 28.511,Y -47.052,Z -242.067,A -90.000,B 90.000,C 0.000} C_DIS
LIN {X 26.138,Y -47.035,Z -242.885,A -90.000,B 90.000,C 0.000} C_DIS
LIN {X 25.427,Y -47.035,Z -243.089,A -90.000,B 90.000,C 0.000} C_DIS
LIN {X 24.912,Y -47.034,Z -243.244,A -90.000,B 90.000,C 0.000} C_DIS
LIN {X 24.655,Y -47.037,Z -243.303,A -90.000,B 90.000,C 0.000} C_DIS
LIN {X 24.478,Y -47.040,Z -243.332,A -90.000,B 90.000,C 0.000} C_DIS
LIN {X 24.340,Y -47.043,Z -243.349,A -90.000,B 90.000,C 0.000} C_DIS
LIN {X 23.928,Y -47.060,Z -243.345,A -90.000,B 90.000,C 0.000} C_DIS
LIN {X 23.623,Y -47.077,Z -243.306,A -90.000,B 90.000,C 0.000} C_DIS
LIN {X 22.954,Y -47.120,Z -243.186,A -90.000,B 90.000,C 0.000} C_DIS
LIN {X 22.817,Y -47.125,Z -243.161,A -90.000,B 90.000,C 0.000} C_DIS
LIN {X 20.973,Y -47.126,Z -242.817,A -90.000,B 90.000,C 0.000} C_DIS
LIN {X 20.639,Y -47.130,Z -242.756,A -90.000,B 90.000,C 0.000} C_DIS
LIN {X 19.963,Y -47.130,Z -242.717,A -90.000,B 90.000,C 0.000} C_DIS
LIN {X 19.586,Y -47.130,Z -242.696,A -90.000,B 90.000,C 0.000} C_DIS
LIN {X 19.449,Y -47.131,Z -242.684,A -90.000,B 90.000,C 0.000} C_DIS
LIN {X 18.995,Y -47.133,Z -242.629,A -90.000,B 90.000,C 0.000} C_DIS
LIN {X 18.911,Y -47.134,Z -242.614,A -90.000,B 90.000,C 0.000} C_DIS
LIN {X 18.462,Y -47.145,Z -242.469,A -90.000,B 90.000,C 0.000} C_DIS
LIN {X 18.364,Y -47.149,Z -242.421,A -90.000,B 90.000,C 0.000} C_DIS
LIN {X 18.233,Y -47.153,Z -242.349,A -90.000,B 90.000,C 0.000} C_DIS
LIN {X 18.070,Y -47.161,Z -242.246,A -90.000,B 90.000,C 0.000} C_DIS
LIN {X 18.012,Y -47.161,Z -242.203,A -90.000,B 90.000,C 0.000} C_DIS
LIN {X 17.906,Y -47.158,Z -242.116,A -90.000,B 90.000,C 0.000} C_DIS
LIN {X 17.755,Y -47.154,Z -241.968,A -90.000,B 90.000,C 0.000} C_DIS
LIN {X 17.539,Y -47.150,Z -241.687,A -90.000,B 90.000,C 0.000} C_DIS
LIN {X 17.188,Y -47.150,Z -241.097,A -90.000,B 90.000,C 0.000} C_DIS
LIN {X 15.728,Y -47.178,Z -238.644,A -90.000,B 90.000,C 0.000} C_DIS
LIN {X 15.494,Y -47.163,Z -238.247,A -90.000,B 90.000,C 0.000} C_DIS
LIN {X 15.385,Y -47.148,Z -238.061,A -90.000,B 90.000,C 0.000} C_DIS
LIN {X 15.308,Y -47.137,Z -237.920,A -90.000,B 90.000,C 0.000} C_DIS
LIN {X 15.255,Y -47.128,Z -237.814,A -90.000,B 90.000,C 0.000} C_DIS
LIN {X 15.232,Y -47.125,Z -237.763,A -90.000,B 90.000,C 0.000} C_DIS
LIN {X 15.091,Y -47.101,Z -237.306,A -90.000,B 90.000,C 0.000} C_DIS
LIN {X 15.076,Y -47.097,Z -237.214,A -90.000,B 90.000,C 0.000} C_DIS
LIN {X 15.015,Y -47.083,Z -236.758,A -90.000,B 90.000,C 0.000} C_DIS
LIN {X 15.001,Y -47.078,Z -236.605,A -90.000,B 90.000,C 0.000} C_DIS
LIN {X 14.990,Y -47.074,Z -236.426,A -90.000,B 90.000,C 0.000} C_DIS
LIN {X 14.991,Y -47.070,Z -236.191,A -90.000,B 90.000,C 0.000} C_DIS
LIN {X 15.000,Y -47.069,Z -236.087,A -90.000,B 90.000,C 0.000} C_DIS
LIN {X 15.011,Y -47.068,Z -236.008,A -90.000,B 90.000,C 0.000} C_DIS
LIN {X 15.025,Y -47.067,Z -235.926,A -90.000,B 90.000,C 0.000} C_DIS
LIN {X 15.914,Y -47.048,Z -231.410,A -90.000,B 90.000,C 0.000} C_DIS
LIN {X 15.984,Y -47.034,Z -231.062,A -90.000,B 90.000,C 0.000} C_DIS
LIN {X 16.034,Y -47.027,Z -230.838,A -90.000,B 90.000,C 0.000} C_DIS
LIN {X 16.077,Y -47.022,Z -230.678,A -90.000,B 90.000,C 0.000} C_DIS
LIN {X 16.204,Y -47.015,Z -230.278,A -90.000,B 90.000,C 0.000} C_DIS
LIN {X 17.458,Y -46.895,Z -226.330,A -90.000,B 90.000,C 0.000} C_DIS
LIN {X 17.525,Y -46.889,Z -226.125,A -90.000,B 90.000,C 0.000} C_DIS
LIN {X 17.565,Y -46.887,Z -226.025,A -90.000,B 90.000,C 0.000} C_DIS
LIN {X 17.881,Y -46.881,Z -225.281,A -90.000,B 90.000,C 0.000} C_DIS
LIN {X 17.940,Y -46.879,Z -225.151,A -90.000,B 90.000,C 0.000} C_DIS
LIN {X 18.685,Y -46.870,Z -223.614,A -90.000,B 90.000,C 0.000} C_DIS
LIN {X 20.361,Y -46.869,Z -220.366,A -90.000,B 90.000,C 0.000} C_DIS
LIN {X 20.481,Y -46.868,Z -220.134,A -90.000,B 90.000,C 0.000} C_DIS
LIN {X 21.006,Y -46.868,Z -219.173,A -90.000,B 90.000,C 0.000} C_DIS
LIN {X 22.456,Y -46.889,Z -216.515,A -90.000,B 90.000,C 0.000} C_DIS
LIN {X 22.946,Y -46.889,Z -215.542,A -90.000,B 90.000,C 0.000} C_DIS
LIN {X 23.102,Y -46.886,Z -215.235,A -90.000,B 90.000,C 0.000} C_DIS
LIN {X 24.177,Y -46.913,Z -213.301,A -90.000,B 90.000,C 0.000} C_DIS
LIN {X 24.731,Y -46.926,Z -212.304,A -90.000,B 90.000,C 0.000} C_DIS
LIN {X 25.283,Y -46.913,Z -211.146,A -90.000,B 90.000,C 0.000} C_DIS
LIN {X 25.560,Y -46.915,Z -210.560,A -90.000,B 90.000,C 0.000} C_DIS
LIN {X 25.617,Y -46.915,Z -210.449,A -90.000,B 90.000,C 0.000} C_DIS
LIN {X 26.524,Y -46.939,Z -208.805,A -90.000,B 90.000,C 0.000} C_DIS
LIN {X 27.173,Y -46.920,Z -207.290,A -90.000,B 90.000,C 0.000} C_DIS
LIN {X 27.612,Y -46.932,Z -206.254,A -90.000,B 90.000,C 0.000} C_DIS
LIN {X 27.685,Y -46.932,Z -206.083,A -90.000,B 90.000,C 0.000} C_DIS
LIN {X 27.740,Y -46.932,Z -205.965,A -90.000,B 90.000,C 0.000} C_DIS
LIN {X 28.107,Y -46.945,Z -205.269,A -90.000,B 90.000,C 0.000} C_DIS
LIN {X 28.537,Y -46.927,Z -204.061,A -90.000,B 90.000,C 0.000} C_DIS
LIN {X 28.993,Y -46.947,Z -202.756,A -90.000,B 90.000,C 0.000} C_DIS
LIN {X 29.031,Y -46.949,Z -202.653,A -90.000,B 90.000,C 0.000} C_DIS
LIN {X 29.262,Y -46.964,Z -202.092,A -90.000,B 90.000,C 0.000} C_DIS
LIN {X 29.358,Y -46.967,Z -201.861,A -90.000,B 90.000,C 0.000} C_DIS
LIN {X 29.403,Y -46.965,Z -201.722,A -90.000,B 90.000,C 0.000} C_DIS
LIN {X 29.646,Y -46.965,Z -201.100,A -90.000,B 90.000,C 0.000} C_DIS
LIN {X 30.565,Y -47.036,Z -198.721,A -90.000,B 90.000,C 0.000} C_DIS
LIN {X 30.662,Y -47.036,Z -198.132,A -90.000,B 90.000,C 0.000} C_DIS
LIN {X 30.715,Y -47.036,Z -197.891,A -90.000,B 90.000,C 0.000} C_DIS
LIN {X 30.797,Y -47.038,Z -197.612,A -90.000,B 90.000,C 0.000} C_DIS
LIN {X 31.517,Y -47.071,Z -195.697,A -90.000,B 90.000,C 0.000} C_DIS
LIN {X 31.599,Y -47.058,Z -195.084,A -90.000,B 90.000,C 0.000} C_DIS
LIN {X 31.687,Y -47.062,Z -194.407,A -90.000,B 90.000,C 0.000} C_DIS
LIN {X 31.700,Y -47.063,Z -194.318,A -90.000,B 90.000,C 0.000} C_DIS
LIN {X 31.728,Y -47.063,Z -194.182,A -90.000,B 90.000,C 0.000} C_DIS
LIN {X 31.777,Y -47.061,Z -193.974,A -90.000,B 90.000,C 0.000} C_DIS
LIN {X 31.873,Y -47.061,Z -193.698,A -90.000,B 90.000,C 0.000} C_DIS
LIN {X 32.323,Y -47.075,Z -192.660,A -90.000,B 90.000,C 0.000} C_DIS
LIN {X 32.442,Y -47.069,Z -192.177,A -90.000,B 90.000,C 0.000} C_DIS
LIN {X 32.807,Y -47.074,Z -190.690,A -90.000,B 90.000,C 0.000} C_DIS
LIN {X 32.849,Y -47.069,Z -190.525,A -90.000,B 90.000,C 0.000} C_DIS
LIN {X 32.877,Y -47.066,Z -190.434,A -90.000,B 90.000,C 0.000} C_DIS
LIN {X 33.019,Y -47.060,Z -190.107,A -90.000,B 90.000,C 0.000} C_DIS
LIN {X 33.104,Y -47.059,Z -189.949,A -90.000,B 90.000,C 0.000} C_DIS
LIN {X 33.156,Y -47.059,Z -189.860,A -90.000,B 90.000,C 0.000} C_DIS
LIN {X 34.474,Y -47.068,Z -187.704,A -90.000,B 90.000,C 0.000} C_DIS
LIN {X 34.550,Y -47.069,Z -187.586,A -90.000,B 90.000,C 0.000} C_DIS
LIN {X 34.980,Y -47.050,Z -186.919,A -90.000,B 90.000,C 0.000} C_DIS
LIN {X 35.214,Y -47.046,Z -186.621,A -90.000,B 90.000,C 0.000} C_DIS
LIN {X 35.302,Y -47.047,Z -186.530,A -90.000,B 90.000,C 0.000} C_DIS
LIN {X 36.322,Y -47.072,Z -185.454,A -90.000,B 90.000,C 0.000} C_DIS
LIN {X 36.449,Y -47.072,Z -185.294,A -90.000,B 90.000,C 0.000} C_DIS
LIN {X 36.648,Y -47.073,Z -185.043,A -90.000,B 90.000,C 0.000} C_DIS
LIN {X 36.916,Y -47.064,Z -184.706,A -90.000,B 90.000,C 0.000} C_DIS
LIN {X 37.277,Y -47.062,Z -184.251,A -90.000,B 90.000,C 0.000} C_DIS
LIN {X 37.416,Y -47.063,Z -184.092,A -90.000,B 90.000,C 0.000} C_DIS
LIN {X 37.578,Y -47.067,Z -183.927,A -90.000,B 90.000,C 0.000} C_DIS
LIN {X 37.995,Y -47.068,Z -183.546,A -90.000,B 90.000,C 0.000} C_DIS
LIN {X 38.436,Y -47.056,Z -183.012,A -90.000,B 90.000,C 0.000} C_DIS
LIN {X 38.648,Y -47.056,Z -182.754,A -90.000,B 90.000,C 0.000} C_DIS
LIN {X 39.209,Y -47.045,Z -182.074,A -90.000,B 90.000,C 0.000} C_DIS
LIN {X 39.316,Y -47.044,Z -181.955,A -90.000,B 90.000,C 0.000} C_DIS
LIN {X 39.451,Y -47.043,Z -181.815,A -90.000,B 90.000,C 0.000} C_DIS
LIN {X 39.548,Y -47.044,Z -181.721,A -90.000,B 90.000,C 0.000} C_DIS
LIN {X 39.604,Y -47.044,Z -181.671,A -90.000,B 90.000,C 0.000} C_DIS
LIN {X 39.858,Y -47.045,Z -181.430,A -90.000,B 90.000,C 0.000} C_DIS
LIN {X 40.965,Y -47.081,Z -180.381,A -90.000,B 90.000,C 0.000} C_DIS
LIN {X 41.314,Y -47.084,Z -179.960,A -90.000,B 90.000,C 0.000} C_DIS
LIN {X 41.421,Y -47.087,Z -179.830,A -90.000,B 90.000,C 0.000} C_DIS
LIN {X 42.165,Y -47.107,Z -178.908,A -90.000,B 90.000,C 0.000} C_DIS
LIN {X 42.633,Y -47.114,Z -178.261,A -90.000,B 90.000,C 0.000} C_DIS
LIN {X 42.995,Y -47.125,Z -177.761,A -90.000,B 90.000,C 0.000} C_DIS
LIN {X 43.106,Y -47.128,Z -177.599,A -90.000,B 90.000,C 0.000} C_DIS
LIN {X 43.368,Y -47.128,Z -177.214,A -90.000,B 90.000,C 0.000} C_DIS
LIN {X 43.901,Y -47.126,Z -176.398,A -90.000,B 90.000,C 0.000} C_DIS
LIN {X 44.474,Y -47.128,Z -175.518,A -90.000,B 90.000,C 0.000} C_DIS
LIN {X 44.555,Y -47.128,Z -175.389,A -90.000,B 90.000,C 0.000} C_DIS
LIN {X 45.073,Y -47.125,Z -174.520,A -90.000,B 90.000,C 0.000} C_DIS
LIN {X 45.841,Y -47.126,Z -173.272,A -90.000,B 90.000,C 0.000} C_DIS
LIN {X 46.264,Y -47.123,Z -172.541,A -90.000,B 90.000,C 0.000} C_DIS
LIN {X 46.369,Y -47.124,Z -172.378,A -90.000,B 90.000,C 0.000} C_DIS
LIN {X 46.421,Y -47.124,Z -172.306,A -90.000,B 90.000,C 0.000} C_DIS
LIN {X 46.514,Y -47.126,Z -172.185,A -90.000,B 90.000,C 0.000} C_DIS
LIN {X 46.588,Y -47.129,Z -172.101,A -90.000,B 90.000,C 0.000} C_DIS
LIN {X 46.723,Y -47.134,Z -171.970,A -90.000,B 90.000,C 0.000} C_DIS
LIN {X 46.859,Y -47.140,Z -171.860,A -90.000,B 90.000,C 0.000} C_DIS
LIN {X 46.987,Y -47.147,Z -171.772,A -90.000,B 90.000,C 0.000} C_DIS
LIN {X 48.232,Y -47.217,Z -170.990,A -90.000,B 90.000,C 0.000} C_DIS
LIN {X 49.022,Y -47.255,Z -170.455,A -90.000,B 90.000,C 0.000} C_DIS
LIN {X 49.363,Y -47.255,Z -170.224,A -90.000,B 90.000,C 0.000} C_DIS
LIN {X 49.778,Y -47.255,Z -169.955,A -90.000,B 90.000,C 0.000} C_DIS
LIN {X 49.975,Y -47.253,Z -169.705,A -90.000,B 90.000,C 0.000} C_DIS
LIN {X 50.315,Y -47.250,Z -169.273,A -90.000,B 90.000,C 0.000} C_DIS
LIN {X 50.408,Y -47.250,Z -169.163,A -90.000,B 90.000,C 0.000} C_DIS
LIN {X 50.476,Y -47.251,Z -169.093,A -90.000,B 90.000,C 0.000} C_DIS
LIN {X 50.747,Y -47.253,Z -168.866,A -90.000,B 90.000,C 0.000} C_DIS
LIN {X 50.957,Y -47.255,Z -168.722,A -90.000,B 90.000,C 0.000} C_DIS
LIN {X 51.116,Y -47.256,Z -168.626,A -90.000,B 90.000,C 0.000} C_DIS
LIN {X 51.166,Y -47.256,Z -168.600,A -90.000,B 90.000,C 0.000} C_DIS
LIN {X 51.388,Y -47.258,Z -168.505,A -90.000,B 90.000,C 0.000} C_DIS
LIN {X 51.488,Y -47.259,Z -168.472,A -90.000,B 90.000,C 0.000} C_DIS
LIN {X 51.606,Y -47.261,Z -168.440,A -90.000,B 90.000,C 0.000} C_DIS
LIN {X 52.003,Y -47.267,Z -168.388,A -90.000,B 90.000,C 0.000} C_DIS
LIN {X 52.003,Y -60.000,Z -168.388,A -90.000,B 90.000,C 0.000} C_DIS
LIN {X 16.531,Y -60.000,Z -243.561,A -90.000,B 90.000,C 0.000} C_DIS
LIN {X 16.531,Y -47.017,Z -243.561,A -90.000,B 90.000,C 0.000} C_DIS
LIN {X 16.362,Y -47.016,Z -243.397,A -90.000,B 90.000,C 0.000} C_DIS
LIN {X 16.181,Y -47.016,Z -243.195,A -90.000,B 90.000,C 0.000} C_DIS
LIN {X 15.957,Y -47.018,Z -242.903,A -90.000,B 90.000,C 0.000} C_DIS
LIN {X 15.824,Y -47.020,Z -242.708,A -90.000,B 90.000,C 0.000} C_DIS
LIN {X 14.384,Y -47.048,Z -240.289,A -90.000,B 90.000,C 0.000} C_DIS
LIN {X 14.145,Y -47.031,Z -239.883,A -90.000,B 90.000,C 0.000} C_DIS
LIN {X 13.674,Y -46.962,Z -239.080,A -90.000,B 90.000,C 0.000} C_DIS
LIN {X 13.569,Y -46.947,Z -238.890,A -90.000,B 90.000,C 0.000} C_DIS
LIN {X 13.480,Y -46.933,Z -238.716,A -90.000,B 90.000,C 0.000} C_DIS
LIN {X 13.435,Y -46.926,Z -238.619,A -90.000,B 90.000,C 0.000} C_DIS
LIN {X 13.376,Y -46.917,Z -238.478,A -90.000,B 90.000,C 0.000} C_DIS
LIN {X 13.335,Y -46.910,Z -238.359,A -90.000,B 90.000,C 0.000} C_DIS
LIN {X 13.194,Y -46.886,Z -237.902,A -90.000,B 90.000,C 0.000} C_DIS
LIN {X 13.164,Y -46.881,Z -237.794,A -90.000,B 90.000,C 0.000} C_DIS
LIN {X 13.129,Y -46.874,Z -237.623,A -90.000,B 90.000,C 0.000} C_DIS
LIN {X 13.115,Y -46.871,Z -237.532,A -90.000,B 90.000,C 0.000} C_DIS
LIN {X 13.048,Y -46.854,Z -237.037,A -90.000,B 90.000,C 0.000} C_DIS
LIN {X 13.035,Y -46.851,Z -236.922,A -90.000,B 90.000,C 0.000} C_DIS
LIN {X 13.018,Y -46.846,Z -236.723,A -90.000,B 90.000,C 0.000} C_DIS
LIN {X 13.004,Y -46.839,Z -236.426,A -90.000,B 90.000,C 0.000} C_DIS
LIN {X 13.005,Y -46.835,Z -236.191,A -90.000,B 90.000,C 0.000} C_DIS
LIN {X 13.010,Y -46.834,Z -236.055,A -90.000,B 90.000,C 0.000} C_DIS
LIN {X 13.021,Y -46.833,Z -235.918,A -90.000,B 90.000,C 0.000} C_DIS
LIN {X 13.042,Y -46.832,Z -235.748,A -90.000,B 90.000,C 0.000} C_DIS
LIN {X 13.068,Y -46.833,Z -235.584,A -90.000,B 90.000,C 0.000} C_DIS
LIN {X 13.110,Y -46.834,Z -235.370,A -90.000,B 90.000,C 0.000} C_DIS
LIN {X 13.205,Y -46.832,Z -234.885,A -90.000,B 90.000,C 0.000} C_DIS
LIN {X 13.415,Y -46.792,Z -233.845,A -90.000,B 90.000,C 0.000} C_DIS
LIN {X 14.069,Y -46.636,Z -230.645,A -90.000,B 90.000,C 0.000} C_DIS
LIN {X 14.141,Y -46.622,Z -230.336,A -90.000,B 90.000,C 0.000} C_DIS
LIN {X 14.208,Y -46.614,Z -230.097,A -90.000,B 90.000,C 0.000} C_DIS
LIN {X 14.325,Y -46.604,Z -229.727,A -90.000,B 90.000,C 0.000} C_DIS
LIN {X 15.492,Y -46.478,Z -226.064,A -90.000,B 90.000,C 0.000} C_DIS
LIN {X 15.665,Y -46.460,Z -225.528,A -90.000,B 90.000,C 0.000} C_DIS
LIN {X 15.706,Y -46.457,Z -225.414,A -90.000,B 90.000,C 0.000} C_DIS
LIN {X 15.746,Y -46.455,Z -225.314,A -90.000,B 90.000,C 0.000} C_DIS
LIN {X 16.012,Y -46.446,Z -224.689,A -90.000,B 90.000,C 0.000} C_DIS
LIN {X 16.059,Y -46.443,Z -224.579,A -90.000,B 90.000,C 0.000} C_DIS
LIN {X 16.158,Y -46.437,Z -224.356,A -90.000,B 90.000,C 0.000} C_DIS
LIN {X 16.932,Y -46.413,Z -222.766,A -90.000,B 90.000,C 0.000} C_DIS
LIN {X 18.756,Y -46.384,Z -219.244,A -90.000,B 90.000,C 0.000} C_DIS
LIN {X 20.051,Y -46.386,Z -216.876,A -90.000,B 90.000,C 0.000} C_DIS
LIN {X 20.723,Y -46.397,Z -215.645,A -90.000,B 90.000,C 0.000} C_DIS
